KUKA KRL program: EPS_2_25694_SR02_A_20251117072413.src

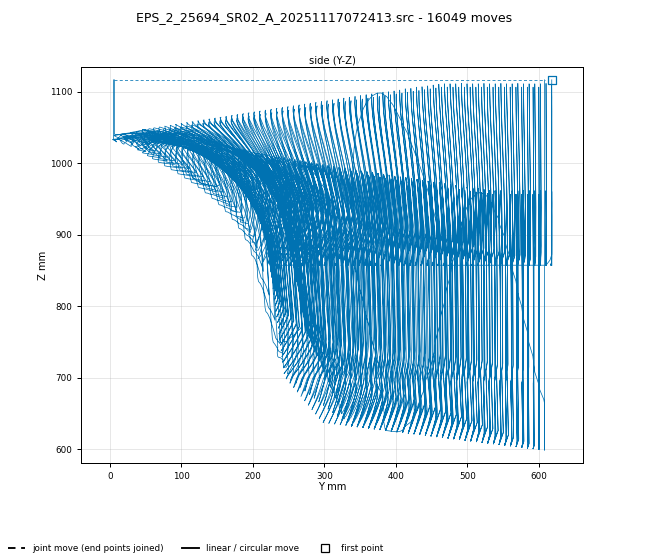
[picture p0: tool path of EPS_2_25694_SR02_A_20251117072413.src, 16049 of 16051 moves have a stored position in this frame; points joined in program order, loops and branches not executed]
&ACCESS RVP
&REL 4
&COMMENT QRS 19112012
&PARAM EDITMASK = *
DEF PART()
EXT BAS (BAS_COMMAND :IN,REAL :IN )
INT I
BAS (#INITMOV,0 )

;KUKA QRS Post kuka4.cps  Date:22-06-2017 !

File_ID=2907

QRS_PRE_INIT()

;Init var - Until changes are made in qrs_pre_init
Outlet_Square_prg=0
Inlet_1_Square_prg=0
Inlet_2_Square_prg=0
Inlet_3_Square_prg=0
Inlet_4_Square_prg=0
Inlet_5_Square_prg=0

Outlet_1={X 0.000, Y 466.000, Z 916.000, B 0.000, E1 0.000 }
Inlet_1={X 0.000, Y 530.840, Z 461.000, B 0.000, E1 112.000 }
Inlet_2={X 0.000, Y 532.280, Z 441.000, B 0.000, E1 197.000 }
Outlet_1_type=381
Inlet_1_type=251
Inlet_2_type=251
;QRS#1=Sidecore dimensions
;QRS#2=375-15" Concrete
;QRS#3=250-10" PVC SDR 35
;QRS#4=250-10" PVC SDR 35
;QRS#5=
;QRS#6=
;QRS#7=
;QRS#8=
;QRS#9=24L PSX-2
;QRS#10=14M PSX
;QRS#11=14M PSX
;QRS#12=
;QRS#13=
;QRS#14=
;QRS#15=
;QRS#16=1220x127x1448 4,75'
;QRS#17=EPS Height
;QRS#18=1106,5
;QRS#19=*
;QRS#20= UPDATED VERSION 22-06-2017
;QRS#21=*
Outlet_Square=0150
Inlet_1_Square=0100
Inlet_2_Square=0100
Inlet_3_Square=0
Inlet_4_Square=0
Inlet_5_Square=0
Mill_Square=1
Outlet_Square_Prg=261
Inlet_1_Square_prg=205
Inlet_2_Square_prg=205

QRS_INIT()

$ADVANCE=5

; T1
PTP {E1 171.09,E2 171.09}
PTP {X 0,Y 618.04,A -85,B 0,C 180,E1 171.09,E2 171.09,E3 0,E4 0,E5 0,E6 0}
QRS_SPEED_INIT()
LIN {X 0,Y 618.04,Z 1116.5,A -85,B 0,C 180,E1 171.09,E2 171.09,E3 0,E4 0,E5 0,E6 0} C_VEL
LIN {X 0,Y 618.04,Z 893.453,A -85,B 0,C 180,E1 171.09,E2 171.09} C_VEL
LIN {X 0,Y 618.04,Z 872.961,A -85,B 0,C 180,E1 171.09,E2 171.09} C_VEL
LIN {X 0,Y 618.039,Z 872.148,A -85,B 0,C 180,E1 171.106,E2 171.106} C_VEL
LIN {X 0,Y 618.037,Z 863.35,A -85,B 0,C 180,E1 171.469,E2 171.469} C_VEL
LIN {X 0,Y 617.988,Z 857.28,A -85,B 0,C 180,E1 171.692,E2 171.692} C_VEL
LIN {X 0,Y 618.064,Z 857.28,A -85,B 0,C 180,E1 171.887,E2 171.887} C_VEL
LIN {X 0,Y 618.025,Z 857.28,A -85,B 0,C 180,E1 174.214,E2 174.214} C_VEL
LIN {X 0,Y 618.042,Z 857.28,A -85,B 0,C 180,E1 178.845,E2 178.845} C_VEL
LIN {X 0,Y 618.069,Z 857.28,A -85,B 0,C 180,E1 183.468,E2 183.468} C_VEL
LIN {X 0,Y 618.042,Z 857.28,A -85,B 0,C 180,E1 188.114,E2 188.114} C_VEL
LIN {X 0,Y 617.972,Z 857.28,A -85,B 0,C 180,E1 192.816,E2 192.816} C_VEL
LIN {X 0,Y 617.962,Z 857.28,A -85,B 0,C 180,E1 197.607,E2 197.607} C_VEL
LIN {X 0,Y 617.779,Z 857.28,A -85,B 0,C 180,E1 198.55,E2 198.55} C_VEL
LIN {X 0,Y 617.956,Z 857.28,A -85,B 0,C 180,E1 202.529,E2 202.529} C_VEL
LIN {X 0,Y 617.453,Z 857.28,A -85,B 0,C 180,E1 205.076,E2 205.076} C_VEL
LIN {X 0,Y 617.89,Z 857.28,A -85,B 0,C 180,E1 207.636,E2 207.636} C_VEL
LIN {X 0,Y 617.381,Z 857.28,A -85,B 0,C 180,E1 210.305,E2 210.305} C_VEL
LIN {X 0,Y 617.848,Z 857.28,A -85,B 0,C 180,E1 212.995,E2 212.995} C_VEL
LIN {X 0,Y 617.72,Z 857.28,A -85,B 0,C 180,E1 214.198,E2 214.198} C_VEL
LIN {X 0,Y 617.794,Z 857.28,A -85,B 0,C 180,E1 218.704,E2 218.704} C_VEL
LIN {X 0,Y 617.454,Z 857.28,A -85,B 0,C 180,E1 221.759,E2 221.759} C_VEL
LIN {X 0,Y 617.88,Z 857.28,A -85,B 0,C 180,E1 224.901,E2 224.901} C_VEL
LIN {X 0,Y 617.78,Z 857.28,A -85,B 0,C 180,E1 228.274,E2 228.274} C_VEL
LIN {X 0,Y 617.552,Z 857.28,A -85,B 0,C 180,E1 231.278,E2 231.278} C_VEL
LIN {X 0,Y 617.574,Z 857.28,A -85,B 0,C 180,E1 231.9,E2 231.9} C_VEL
LIN {X 0,Y 617.805,Z 857.28,A -85,B 0,C 180,E1 234.201,E2 234.201} C_VEL
LIN {X 0,Y 617.346,Z 857.28,A -85,B 0,C 180,E1 236.975,E2 236.975} C_VEL
LIN {X 0,Y 617.903,Z 857.28,A -85,B 0,C 180,E1 239.723,E2 239.723} C_VEL
LIN {X 0,Y 617.426,Z 857.28,A -85,B 0,C 180,E1 242.341,E2 242.341} C_VEL
LIN {X 0,Y 617.95,Z 857.28,A -85,B 0,C 180,E1 244.946,E2 244.946} C_VEL
LIN {X 0,Y 617.971,Z 857.28,A -85,B 0,C 180,E1 247.993,E2 247.993} C_VEL
LIN {X 0,Y 617.845,Z 857.28,A -85,B 0,C 180,E1 248.248,E2 248.248} C_VEL
LIN {X 0,Y 616.597,Z 857.28,A -85,B 0,C 180,E1 248.461,E2 248.461} C_VEL
LIN {X 0,Y 617.498,Z 860.533,A -85,B 0,C 180,E1 248.542,E2 248.542} C_VEL
LIN {X 0,Y 617.689,Z 861.463,A -85,B 0,C 180,E1 248.56,E2 248.56} C_VEL
LIN {X 0,Y 617.924,Z 919.311,A -85,B 0,C 180,E1 249.277,E2 249.277} C_VEL
LIN {X 0,Y 618.001,Z 930.791,A -85,B 0,C 180,E1 249.459,E2 249.459} C_VEL
LIN {X 0,Y 617.956,Z 939.703,A -85,B 0,C 180,E1 249.638,E2 249.638} C_VEL
LIN {X 0,Y 617.868,Z 948.851,A -85,B 0,C 180,E1 249.859,E2 249.859} C_VEL
LIN {X 0,Y 617.969,Z 959.233,A -85,B 0,C 180,E1 250.169,E2 250.169} C_VEL
LIN {X 0,Y 617.951,Z 969.224,A -85,B 0,C 180,E1 250.516,E2 250.516} C_VEL
LIN {X 0,Y 617.933,Z 976.981,A -85,B 0,C 180,E1 250.818,E2 250.818} C_VEL
LIN {X 0,Y 617.992,Z 986.692,A -85,B 0,C 180,E1 251.252,E2 251.252} C_VEL
LIN {X 0,Y 618.003,Z 996.669,A -85,B 0,C 180,E1 251.755,E2 251.755} C_VEL
LIN {X 0,Y 617.953,Z 1005.465,A -85,B 0,C 180,E1 252.248,E2 252.248} C_VEL
LIN {X 0,Y 617.994,Z 1014.291,A -85,B 0,C 180,E1 252.801,E2 252.801} C_VEL
LIN {X 0,Y 617.978,Z 1023.074,A -85,B 0,C 180,E1 253.409,E2 253.409} C_VEL
LIN {X 0,Y 617.993,Z 1031.008,A -85,B 0,C 180,E1 254.015,E2 254.015} C_VEL
LIN {X 0,Y 617.98,Z 1038.115,A -85,B 0,C 180,E1 254.606,E2 254.606} C_VEL
LIN {X 0,Y 617.953,Z 1043.662,A -85,B 0,C 180,E1 255.101,E2 255.101} C_VEL
LIN {X 0,Y 617.981,Z 1051.279,A -85,B 0,C 180,E1 255.848,E2 255.848} C_VEL
LIN {X 0,Y 618.005,Z 1056.878,A -85,B 0,C 180,E1 256.443,E2 256.443} C_VEL
LIN {X 0,Y 617.937,Z 1063.299,A -85,B 0,C 180,E1 257.184,E2 257.184} C_VEL
LIN {X 0,Y 617.922,Z 1069.145,A -85,B 0,C 180,E1 257.923,E2 257.923} C_VEL
LIN {X 0,Y 617.97,Z 1074.465,A -85,B 0,C 180,E1 258.661,E2 258.661} C_VEL
LIN {X 0,Y 617.959,Z 1080.218,A -85,B 0,C 180,E1 259.544,E2 259.544} C_VEL
LIN {X 0,Y 617.879,Z 1084.857,A -85,B 0,C 180,E1 260.327,E2 260.327} C_VEL
LIN {X 0,Y 617.887,Z 1089.451,A -85,B 0,C 180,E1 261.196,E2 261.196} C_VEL
LIN {X 0,Y 617.977,Z 1093.733,A -85,B 0,C 180,E1 262.119,E2 262.119} C_VEL
LIN {X 0,Y 617.893,Z 1096.689,A -85,B 0,C 180,E1 262.817,E2 262.817} C_VEL
LIN {X 0,Y 617.823,Z 1100.1,A -85,B 0,C 180,E1 263.747,E2 263.747} C_VEL
LIN {X 0,Y 617.905,Z 1102.963,A -85,B 0,C 180,E1 264.677,E2 264.677} C_VEL
LIN {X 0,Y 617.95,Z 1105.345,A -85,B 0,C 180,E1 265.605,E2 265.605} C_VEL
LIN {X 0,Y 617.834,Z 1107.293,A -85,B 0,C 180,E1 266.531,E2 266.531} C_VEL
LIN {X 0,Y 617.839,Z 1108.744,A -85,B 0,C 180,E1 267.457,E2 267.457} C_VEL
LIN {X 0,Y 617.944,Z 1110.042,A -85,B 0,C 180,E1 268.845,E2 268.845} C_VEL
LIN {X 0,Y 617.878,Z 1110.288,A -85,B 0,C 180,E1 269.307,E2 269.307} C_VEL
LIN {X 0,Y 617.832,Z 1110.409,A -85,B 0,C 180,E1 270.231,E2 270.231} C_VEL
LIN {X 0,Y 617.902,Z 1110.053,A -85,B 0,C 180,E1 271.156,E2 271.156} C_VEL
LIN {X 0,Y 617.951,Z 1109.26,A -85,B 0,C 180,E1 272.08,E2 272.08} C_VEL
LIN {X 0,Y 617.822,Z 1107.296,A -85,B 0,C 180,E1 273.469,E2 273.469} C_VEL
LIN {X 0,Y 617.899,Z 1105.359,A -85,B 0,C 180,E1 274.395,E2 274.395} C_VEL
LIN {X 0,Y 617.943,Z 1102.953,A -85,B 0,C 180,E1 275.323,E2 275.323} C_VEL
LIN {X 0,Y 617.836,Z 1100.097,A -85,B 0,C 180,E1 276.253,E2 276.253} C_VEL
LIN {X 0,Y 617.864,Z 1096.696,A -85,B 0,C 180,E1 277.183,E2 277.183} C_VEL
LIN {X 0,Y 617.981,Z 1091.704,A -85,B 0,C 180,E1 278.334,E2 278.334} C_VEL
LIN {X 0,Y 617.877,Z 1086.888,A -85,B 0,C 180,E1 279.301,E2 279.301} C_VEL
LIN {X 0,Y 617.884,Z 1082.576,A -85,B 0,C 180,E1 280.072,E2 280.072} C_VEL
LIN {X 0,Y 617.947,Z 1078.418,A -85,B 0,C 180,E1 280.751,E2 280.751} C_VEL
LIN {X 0,Y 617.962,Z 1072.408,A -85,B 0,C 180,E1 281.634,E2 281.634} C_VEL
LIN {X 0,Y 617.908,Z 1065.701,A -85,B 0,C 180,E1 282.521,E2 282.521} C_VEL
LIN {X 0,Y 617.947,Z 1059.514,A -85,B 0,C 180,E1 283.261,E2 283.261} C_VEL
LIN {X 0,Y 617.996,Z 1054.147,A -85,B 0,C 180,E1 283.854,E2 283.854} C_VEL
LIN {X 0,Y 617.97,Z 1046.794,A -85,B 0,C 180,E1 284.6,E2 284.6} C_VEL
LIN {X 0,Y 617.961,Z 1040.369,A -85,B 0,C 180,E1 285.198,E2 285.198} C_VEL
LIN {X 0,Y 617.985,Z 1032.107,A -85,B 0,C 180,E1 285.897,E2 285.897} C_VEL
LIN {X 0,Y 617.995,Z 1024.024,A -85,B 0,C 180,E1 286.521,E2 286.521} C_VEL
LIN {X 0,Y 617.984,Z 1016.498,A -85,B 0,C 180,E1 287.052,E2 287.052} C_VEL
LIN {X 0,Y 617.987,Z 1009.682,A -85,B 0,C 180,E1 287.495,E2 287.495} C_VEL
LIN {X 0,Y 617.943,Z 1001.121,A -85,B 0,C 180,E1 288.003,E2 288.003} C_VEL
LIN {X 0,Y 617.999,Z 992.467,A -85,B 0,C 180,E1 288.464,E2 288.464} C_VEL
LIN {X 0,Y 618.009,Z 982.893,A -85,B 0,C 180,E1 288.921,E2 288.921} C_VEL
LIN {X 0,Y 617.967,Z 973.713,A -85,B 0,C 180,E1 289.311,E2 289.311} C_VEL
LIN {X 0,Y 617.906,Z 965.71,A -85,B 0,C 180,E1 289.616,E2 289.616} C_VEL
LIN {X 0,Y 618.002,Z 954.078,A -85,B 0,C 180,E1 289.987,E2 289.987} C_VEL
LIN {X 0,Y 617.983,Z 944.339,A -85,B 0,C 180,E1 290.251,E2 290.251} C_VEL
LIN {X 0,Y 617.847,Z 934.408,A -85,B 0,C 180,E1 290.477,E2 290.477} C_VEL
LIN {X 0,Y 617.928,Z 924.756,A -85,B 0,C 180,E1 290.644,E2 290.644} C_VEL
LIN {X 0,Y 617.881,Z 903.608,A -85,B 0,C 180,E1 290.919,E2 290.919} C_VEL
LIN {X 0,Y 617.753,Z 864.651,A -85,B 0,C 180,E1 291.399,E2 291.399} C_VEL
LIN {X 0,Y 617.582,Z 861.01,A -85,B 0,C 180,E1 291.45,E2 291.45} C_VEL
LIN {X 0,Y 616.602,Z 857.28,A -85,B 0,C 180,E1 291.54,E2 291.54} C_VEL
LIN {X 0,Y 618.005,Z 857.28,A -85,B 0,C 180,E1 291.926,E2 291.926} C_VEL
LIN {X 0,Y 618.025,Z 857.28,A -85,B 0,C 180,E1 292.526,E2 292.526} C_VEL
LIN {X 0,Y 617.436,Z 857.28,A -85,B 0,C 180,E1 295.077,E2 295.077} C_VEL
LIN {X 0,Y 617.88,Z 857.28,A -85,B 0,C 180,E1 297.637,E2 297.637} C_VEL
LIN {X 0,Y 617.376,Z 857.28,A -85,B 0,C 180,E1 300.306,E2 300.306} C_VEL
LIN {X 0,Y 617.847,Z 857.28,A -85,B 0,C 180,E1 302.995,E2 302.995} C_VEL
LIN {X 0,Y 617.71,Z 857.28,A -85,B 0,C 180,E1 304.197,E2 304.197} C_VEL
LIN {X 0,Y 617.806,Z 857.28,A -85,B 0,C 180,E1 308.703,E2 308.703} C_VEL
LIN {X 0,Y 617.453,Z 857.28,A -85,B 0,C 180,E1 311.759,E2 311.759} C_VEL
LIN {X 0,Y 617.865,Z 857.28,A -85,B 0,C 180,E1 314.902,E2 314.902} C_VEL
LIN {X 0,Y 617.768,Z 857.28,A -85,B 0,C 180,E1 318.275,E2 318.275} C_VEL
LIN {X 0,Y 617.555,Z 857.28,A -85,B 0,C 180,E1 321.279,E2 321.279} C_VEL
LIN {X 0,Y 617.591,Z 857.28,A -85,B 0,C 180,E1 321.898,E2 321.898} C_VEL
LIN {X 0,Y 617.836,Z 857.28,A -85,B 0,C 180,E1 324.203,E2 324.203} C_VEL
LIN {X 0,Y 617.346,Z 857.28,A -85,B 0,C 180,E1 326.975,E2 326.975} C_VEL
LIN {X 0,Y 617.862,Z 857.28,A -85,B 0,C 180,E1 329.721,E2 329.721} C_VEL
LIN {X 0,Y 617.414,Z 857.28,A -85,B 0,C 180,E1 332.341,E2 332.341} C_VEL
LIN {X 0,Y 617.92,Z 857.28,A -85,B 0,C 180,E1 334.944,E2 334.944} C_VEL
LIN {X 0,Y 617.455,Z 857.28,A -85,B 0,C 180,E1 337.452,E2 337.452} C_VEL
LIN {X 0,Y 617.949,Z 857.28,A -85,B 0,C 180,E1 339.951,E2 339.951} C_VEL
LIN {X 0,Y 618.039,Z 857.28,A -85,B 0,C 180,E1 343.632,E2 343.632} C_VEL
LIN {X 0,Y 618.002,Z 857.28,A -85,B 0,C 180,E1 349.544,E2 349.544} C_VEL
LIN {X 0,Y 618.032,Z 857.28,A -85,B 0,C 180,E1 354.214,E2 354.214} C_VEL
LIN {X 0,Y 618.053,Z 857.28,A -85,B 0,C 180,E1 358.845,E2 358.845} C_VEL
LIN {X 0,Y 618.057,Z 857.28,A -85,B 0,C 180,E1 363.468,E2 363.468} C_VEL
LIN {X 0,Y 618.041,Z 857.28,A -85,B 0,C 180,E1 368.114,E2 368.114} C_VEL
LIN {X 0,Y 617.985,Z 857.28,A -85,B 0,C 180,E1 372.815,E2 372.815} C_VEL
LIN {X 0,Y 617.978,Z 857.28,A -85,B 0,C 180,E1 377.606,E2 377.606} C_VEL
LIN {X 0,Y 617.784,Z 857.28,A -85,B 0,C 180,E1 378.551,E2 378.551} C_VEL
LIN {X 0,Y 617.941,Z 857.28,A -85,B 0,C 180,E1 382.529,E2 382.529} C_VEL
LIN {X 0,Y 617.448,Z 857.28,A -85,B 0,C 180,E1 385.076,E2 385.076} C_VEL
LIN {X 0,Y 617.897,Z 857.28,A -85,B 0,C 180,E1 387.636,E2 387.636} C_VEL
LIN {X 0,Y 617.383,Z 857.28,A -85,B 0,C 180,E1 390.305,E2 390.305} C_VEL
LIN {X 0,Y 617.849,Z 857.28,A -85,B 0,C 180,E1 392.995,E2 392.995} C_VEL
LIN {X 0,Y 617.708,Z 857.28,A -85,B 0,C 180,E1 394.196,E2 394.196} C_VEL
LIN {X 0,Y 617.785,Z 857.28,A -85,B 0,C 180,E1 398.704,E2 398.704} C_VEL
LIN {X 0,Y 617.446,Z 857.28,A -85,B 0,C 180,E1 401.76,E2 401.76} C_VEL
LIN {X 0,Y 617.879,Z 857.28,A -85,B 0,C 180,E1 404.901,E2 404.901} C_VEL
LIN {X 0,Y 617.763,Z 857.28,A -85,B 0,C 180,E1 408.276,E2 408.276} C_VEL
LIN {X 0,Y 617.554,Z 857.28,A -85,B 0,C 180,E1 411.278,E2 411.278} C_VEL
LIN {X 0,Y 617.581,Z 857.28,A -85,B 0,C 180,E1 411.9,E2 411.9} C_VEL
LIN {X 0,Y 617.842,Z 857.28,A -85,B 0,C 180,E1 414.204,E2 414.204} C_VEL
LIN {X 0,Y 618.036,Z 857.28,A -85,B 0,C 180,E1 418.887,E2 418.887} C_VEL
LIN {X 0,Y 618.021,Z 857.28,A -85,B 0,C 180,E1 419.078,E2 419.078} C_VEL
LIN {X 0,Y 617.565,Z 857.357,A -85,B 0,C 180,E1 419.213,E2 419.213} C_VEL
LIN {X 0,Y 617.922,Z 866.552,A -85,B 0,C 180,E1 419.562,E2 419.562} C_VEL
LIN {X 0,Y 617.999,Z 875.408,A -85,B 0,C 180,E1 419.958,E2 419.958} C_VEL
LIN {X 0,Y 617.995,Z 884.21,A -85,B 0,C 180,E1 420.411,E2 420.411} C_VEL
LIN {X 0,Y 618.021,Z 891.714,A -85,B 0,C 180,E1 420.859,E2 420.859} C_VEL
LIN {X 0,Y 618.016,Z 898.437,A -85,B 0,C 180,E1 421.312,E2 421.312} C_VEL
LIN {X 0,Y 618.01,Z 905.925,A -85,B 0,C 180,E1 421.877,E2 421.877} C_VEL
LIN {X 0,Y 617.989,Z 913.549,A -85,B 0,C 180,E1 422.532,E2 422.532} C_VEL
LIN {X 0,Y 617.986,Z 920.183,A -85,B 0,C 180,E1 423.181,E2 423.181} C_VEL
LIN {X 0,Y 617.987,Z 927.401,A -85,B 0,C 180,E1 423.987,E2 423.987} C_VEL
LIN {X 0,Y 617.977,Z 932.435,A -85,B 0,C 180,E1 424.627,E2 424.627} C_VEL
LIN {X 0,Y 617.963,Z 937.67,A -85,B 0,C 180,E1 425.376,E2 425.376} C_VEL
LIN {X 0,Y 617.994,Z 942.305,A -85,B 0,C 180,E1 426.144,E2 426.144} C_VEL
LIN {X 0,Y 617.943,Z 946.382,A -85,B 0,C 180,E1 426.92,E2 426.92} C_VEL
LIN {X 0,Y 617.93,Z 950.266,A -85,B 0,C 180,E1 427.783,E2 427.783} C_VEL
LIN {X 0,Y 617.999,Z 953.633,A -85,B 0,C 180,E1 428.718,E2 428.718} C_VEL
LIN {X 0,Y 617.953,Z 955.499,A -85,B 0,C 180,E1 429.335,E2 429.335} C_VEL
LIN {X 0,Y 617.897,Z 957.055,A -85,B 0,C 180,E1 429.95,E2 429.95} C_VEL
LIN {X 0,Y 617.918,Z 958.426,A -85,B 0,C 180,E1 430.644,E2 430.644} C_VEL
LIN {X 0,Y 617.988,Z 959.481,A -85,B 0,C 180,E1 431.393,E2 431.393} C_VEL
LIN {X 0,Y 617.929,Z 960.308,A -85,B 0,C 180,E1 432.392,E2 432.392} C_VEL
LIN {X 0,Y 617.908,Z 960.363,A -85,B 0,C 180,E1 433.299,E2 433.299} C_VEL
LIN {X 0,Y 617.931,Z 960.207,A -85,B 0,C 180,E1 433.707,E2 433.707} C_VEL
LIN {X 0,Y 617.953,Z 959.156,A -85,B 0,C 180,E1 434.802,E2 434.802} C_VEL
LIN {X 0,Y 617.917,Z 958.206,A -85,B 0,C 180,E1 435.399,E2 435.399} C_VEL
LIN {X 0,Y 617.92,Z 956.973,A -85,B 0,C 180,E1 435.995,E2 435.995} C_VEL
LIN {X 0,Y 617.963,Z 955.452,A -85,B 0,C 180,E1 436.591,E2 436.591} C_VEL
LIN {X 0,Y 617.974,Z 952.698,A -85,B 0,C 180,E1 437.48,E2 437.48} C_VEL
LIN {X 0,Y 617.922,Z 950.503,A -85,B 0,C 180,E1 438.071,E2 438.071} C_VEL
LIN {X 0,Y 617.922,Z 947.977,A -85,B 0,C 180,E1 438.66,E2 438.66} C_VEL
LIN {X 0,Y 617.993,Z 943.521,A -85,B 0,C 180,E1 439.544,E2 439.544} C_VEL
LIN {X 0,Y 617.983,Z 939.081,A -85,B 0,C 180,E1 440.309,E2 440.309} C_VEL
LIN {X 0,Y 617.958,Z 933.399,A -85,B 0,C 180,E1 441.154,E2 441.154} C_VEL
LIN {X 0,Y 617.993,Z 927.705,A -85,B 0,C 180,E1 441.886,E2 441.886} C_VEL
LIN {X 0,Y 618.001,Z 921.58,A -85,B 0,C 180,E1 442.585,E2 442.585} C_VEL
LIN {X 0,Y 617.982,Z 915.8,A -85,B 0,C 180,E1 443.167,E2 443.167} C_VEL
LIN {X 0,Y 618.005,Z 909.346,A -85,B 0,C 180,E1 443.749,E2 443.749} C_VEL
LIN {X 0,Y 618.016,Z 902.149,A -85,B 0,C 180,E1 444.33,E2 444.33} C_VEL
LIN {X 0,Y 618.029,Z 893.855,A -85,B 0,C 180,E1 444.91,E2 444.91} C_VEL
LIN {X 0,Y 618.019,Z 886.367,A -85,B 0,C 180,E1 445.374,E2 445.374} C_VEL
LIN {X 0,Y 618.034,Z 877.771,A -85,B 0,C 180,E1 445.837,E2 445.837} C_VEL
LIN {X 0,Y 618.041,Z 868.943,A -85,B 0,C 180,E1 446.243,E2 446.243} C_VEL
LIN {X 0,Y 618.015,Z 860.032,A -85,B 0,C 180,E1 446.594,E2 446.594} C_VEL
LIN {X 0,Y 617.985,Z 857.28,A -85,B 0,C 180,E1 446.693,E2 446.693} C_VEL
LIN {X 0,Y 618.049,Z 857.28,A -85,B 0,C 180,E1 447.468,E2 447.468} C_VEL
LIN {X 0,Y 617.305,Z 857.28,A -85,B 0,C 180,E1 451.157,E2 451.157} C_VEL
LIN {X 0,Y 618.059,Z 857.28,A -85,B 0,C 180,E1 453.468,E2 453.468} C_VEL
LIN {X 0,Y 618.052,Z 857.28,A -85,B 0,C 180,E1 458.114,E2 458.114} C_VEL
LIN {X 0,Y 618.016,Z 857.28,A -85,B 0,C 180,E1 462.815,E2 462.815} C_VEL
LIN {X 0,Y 617.938,Z 857.28,A -85,B 0,C 180,E1 467.607,E2 467.607} C_VEL
LIN {X 0,Y 617.759,Z 857.28,A -85,B 0,C 180,E1 468.544,E2 468.544} C_VEL
LIN {X 0,Y 617.93,Z 857.28,A -85,B 0,C 180,E1 472.53,E2 472.53} C_VEL
LIN {X 0,Y 617.424,Z 857.28,A -85,B 0,C 180,E1 475.077,E2 475.077} C_VEL
LIN {X 0,Y 617.857,Z 857.28,A -85,B 0,C 180,E1 477.638,E2 477.638} C_VEL
LIN {X 0,Y 617.361,Z 857.28,A -85,B 0,C 180,E1 480.306,E2 480.306} C_VEL
LIN {X 0,Y 617.851,Z 857.28,A -85,B 0,C 180,E1 482.995,E2 482.995} C_VEL
LIN {X 0,Y 617.718,Z 857.28,A -85,B 0,C 180,E1 484.198,E2 484.198} C_VEL
LIN {X 0,Y 617.747,Z 857.28,A -85,B 0,C 180,E1 488.707,E2 488.707} C_VEL
LIN {X 0,Y 617.425,Z 857.28,A -85,B 0,C 180,E1 491.762,E2 491.762} C_VEL
LIN {X 0,Y 617.878,Z 857.28,A -85,B 0,C 180,E1 494.901,E2 494.901} C_VEL
LIN {X 0,Y 617.786,Z 857.28,A -85,B 0,C 180,E1 498.273,E2 498.273} C_VEL
LIN {X 0,Y 617.488,Z 857.28,A -85,B 0,C 180,E1 501.274,E2 501.274} C_VEL
LIN {X 0,Y 617.755,Z 857.299,A -85,B 0,C 180,E1 504.216,E2 504.216} C_VEL
LIN {X 0,Y 617.946,Z 867.414,A -85,B 0,C 180,E1 504.599,E2 504.599} C_VEL
LIN {X 0,Y 617.985,Z 875.042,A -85,B 0,C 180,E1 504.94,E2 504.94} C_VEL
LIN {X 0,Y 618.02,Z 883.242,A -85,B 0,C 180,E1 505.36,E2 505.36} C_VEL
LIN {X 0,Y 618.032,Z 892.212,A -85,B 0,C 180,E1 505.892,E2 505.892} C_VEL
LIN {X 0,Y 617.997,Z 899.299,A -85,B 0,C 180,E1 506.373,E2 506.373} C_VEL
LIN {X 0,Y 618.002,Z 905.644,A -85,B 0,C 180,E1 506.855,E2 506.855} C_VEL
LIN {X 0,Y 618.008,Z 913.37,A -85,B 0,C 180,E1 507.515,E2 507.515} C_VEL
LIN {X 0,Y 617.992,Z 919.727,A -85,B 0,C 180,E1 508.134,E2 508.134} C_VEL
LIN {X 0,Y 617.968,Z 926.591,A -85,B 0,C 180,E1 508.887,E2 508.887} C_VEL
LIN {X 0,Y 617.959,Z 931.93,A -85,B 0,C 180,E1 509.559,E2 509.559} C_VEL
LIN {X 0,Y 617.992,Z 937.196,A -85,B 0,C 180,E1 510.307,E2 510.307} C_VEL
LIN {X 0,Y 617.969,Z 941.404,A -85,B 0,C 180,E1 510.982,E2 510.982} C_VEL
LIN {X 0,Y 617.919,Z 945.817,A -85,B 0,C 180,E1 511.802,E2 511.802} C_VEL
LIN {X 0,Y 617.987,Z 949.867,A -85,B 0,C 180,E1 512.694,E2 512.694} C_VEL
LIN {X 0,Y 617.938,Z 953.473,A -85,B 0,C 180,E1 513.663,E2 513.663} C_VEL
LIN {X 0,Y 617.908,Z 955.428,A -85,B 0,C 180,E1 514.304,E2 514.304} C_VEL
LIN {X 0,Y 617.954,Z 957.484,A -85,B 0,C 180,E1 515.155,E2 515.155} C_VEL
LIN {X 0,Y 618.001,Z 958.389,A -85,B 0,C 180,E1 515.636,E2 515.636} C_VEL
LIN {X 0,Y 617.94,Z 959.543,A -85,B 0,C 180,E1 516.434,E2 516.434} C_VEL
LIN {X 0,Y 617.921,Z 960.327,A -85,B 0,C 180,E1 517.47,E2 517.47} C_VEL
LIN {X 0,Y 617.975,Z 960.393,A -85,B 0,C 180,E1 518.096,E2 518.096} C_VEL
LIN {X 0,Y 617.968,Z 960.189,A -85,B 0,C 180,E1 518.717,E2 518.717} C_VEL
LIN {X 0,Y 617.943,Z 959.71,A -85,B 0,C 180,E1 519.335,E2 519.335} C_VEL
LIN {X 0,Y 617.929,Z 958.95,A -85,B 0,C 180,E1 519.951,E2 519.951} C_VEL
LIN {X 0,Y 617.992,Z 957.697,A -85,B 0,C 180,E1 520.652,E2 520.652} C_VEL
LIN {X 0,Y 617.962,Z 955.964,A -85,B 0,C 180,E1 521.4,E2 521.4} C_VEL
LIN {X 0,Y 617.917,Z 954.689,A -85,B 0,C 180,E1 521.87,E2 521.87} C_VEL
LIN {X 0,Y 617.91,Z 953.019,A -85,B 0,C 180,E1 522.392,E2 522.392} C_VEL
LIN {X 0,Y 617.957,Z 949.943,A -85,B 0,C 180,E1 523.2,E2 523.2} C_VEL
LIN {X 0,Y 617.982,Z 946.308,A -85,B 0,C 180,E1 524.003,E2 524.003} C_VEL
LIN {X 0,Y 617.988,Z 942.107,A -85,B 0,C 180,E1 524.803,E2 524.803} C_VEL
LIN {X 0,Y 617.96,Z 938.532,A -85,B 0,C 180,E1 525.4,E2 525.4} C_VEL
LIN {X 0,Y 617.959,Z 933.465,A -85,B 0,C 180,E1 526.145,E2 526.145} C_VEL
LIN {X 0,Y 617.998,Z 927.679,A -85,B 0,C 180,E1 526.889,E2 526.889} C_VEL
LIN {X 0,Y 617.992,Z 921.164,A -85,B 0,C 180,E1 527.629,E2 527.629} C_VEL
LIN {X 0,Y 617.991,Z 915.241,A -85,B 0,C 180,E1 528.219,E2 528.219} C_VEL
LIN {X 0,Y 618.018,Z 908.638,A -85,B 0,C 180,E1 528.809,E2 528.809} C_VEL
LIN {X 0,Y 618.03,Z 900.192,A -85,B 0,C 180,E1 529.471,E2 529.471} C_VEL
LIN {X 0,Y 618.017,Z 893.812,A -85,B 0,C 180,E1 529.913,E2 529.913} C_VEL
LIN {X 0,Y 618.003,Z 886.379,A -85,B 0,C 180,E1 530.374,E2 530.374} C_VEL
LIN {X 0,Y 618.037,Z 877.84,A -85,B 0,C 180,E1 530.834,E2 530.834} C_VEL
LIN {X 0,Y 618.039,Z 872.148,A -85,B 0,C 180,E1 531.106,E2 531.106} C_VEL
LIN {X 0,Y 615.518,Z 864.313,A -85,B 0,C 180,E1 531.544,E2 531.544} C_VEL
LIN {X 0,Y 610.896,Z 858.156,A -85,B 0,C 180,E1 532.238,E2 532.238} C_VEL
LIN {X 0,Y 610.06,Z 857.28,A -85,B 0,C 180,E1 532.633,E2 532.633} C_VEL
LIN {X 0,Y 610.057,Z 857.28,A -85,B 0,C 180,E1 538.597,E2 538.597} C_VEL
LIN {X 0,Y 609.894,Z 857.28,A -85,B 0,C 180,E1 544.287,E2 544.287} C_VEL
LIN {X 0,Y 609.957,Z 857.28,A -85,B 0,C 180,E1 548.58,E2 548.58} C_VEL
LIN {X 0,Y 610.038,Z 857.28,A -85,B 0,C 180,E1 552.92,E2 552.92} C_VEL
LIN {X 0,Y 609.816,Z 857.28,A -85,B 0,C 180,E1 558.841,E2 558.841} C_VEL
LIN {X 0,Y 609.758,Z 857.28,A -85,B 0,C 180,E1 563.418,E2 563.418} C_VEL
LIN {X 0,Y 609.804,Z 857.28,A -85,B 0,C 180,E1 568.155,E2 568.155} C_VEL
LIN {X 0,Y 609.954,Z 857.28,A -85,B 0,C 180,E1 573.105,E2 573.105} C_VEL
LIN {X 0,Y 609.619,Z 857.28,A -85,B 0,C 180,E1 579.653,E2 579.653} C_VEL
LIN {X 0,Y 609.739,Z 857.28,A -85,B 0,C 180,E1 585.951,E2 585.951} C_VEL
LIN {X 0,Y 609.56,Z 857.28,A -85,B 0,C 180,E1 590.353,E2 590.353} C_VEL
LIN {X 0,Y 609.597,Z 857.28,A -85,B 0,C 180,E1 595.163,E2 595.163} C_VEL
LIN {X 0,Y 609.798,Z 857.28,A -85,B 0,C 180,E1 600.338,E2 600.338} C_VEL
LIN {X 0,Y 610.046,Z 857.28,A -85,B 0,C 180,E1 605.044,E2 605.044} C_VEL
LIN {X 0,Y 609.377,Z 857.28,A -85,B 0,C 180,E1 608.167,E2 608.167} C_VEL
LIN {X 0,Y 610.37,Z 873.803,A -85,B 0,C 180,E1 608.443,E2 608.443} C_VEL
LIN {X 0,Y 610.561,Z 938.64,A -85,B 0,C 180,E1 609.354,E2 609.354} C_VEL
LIN {X 0,Y 610.451,Z 972.232,A -85,B 0,C 180,E1 610.384,E2 610.384} C_VEL
LIN {X 0,Y 610.386,Z 1004.124,A -85,B 0,C 180,E1 611.937,E2 611.937} C_VEL
LIN {X 0,Y 610.297,Z 1033.24,A -85,B 0,C 180,E1 613.979,E2 613.979} C_VEL
LIN {X 0,Y 610.237,Z 1058.073,A -85,B 0,C 180,E1 616.367,E2 616.367} C_VEL
LIN {X 0,Y 610.16,Z 1078.846,A -85,B 0,C 180,E1 619.094,E2 619.094} C_VEL
LIN {X 0,Y 610.159,Z 1095.118,A -85,B 0,C 180,E1 622.156,E2 622.156} C_VEL
LIN {X 0,Y 610.1,Z 1104.988,A -85,B 0,C 180,E1 625.018,E2 625.018} C_VEL
LIN {X 0,Y 610,Z 1109.397,A -85,B 0,C 180,E1 627.155,E2 627.155} C_VEL
LIN {X 0,Y 610.019,Z 1111.5,A -85,B 0,C 180,E1 630.001,E2 630.001} C_VEL
LIN {X 0,Y 610.048,Z 1109.396,A -85,B 0,C 180,E1 632.846,E2 632.846} C_VEL
LIN {X 0,Y 610.051,Z 1101.844,A -85,B 0,C 180,E1 636.056,E2 636.056} C_VEL
LIN {X 0,Y 610.116,Z 1090.12,A -85,B 0,C 180,E1 638.923,E2 638.923} C_VEL
LIN {X 0,Y 610.172,Z 1072.662,A -85,B 0,C 180,E1 641.813,E2 641.813} C_VEL
LIN {X 0,Y 610.233,Z 1050.188,A -85,B 0,C 180,E1 644.477,E2 644.477} C_VEL
LIN {X 0,Y 610.332,Z 1022.478,A -85,B 0,C 180,E1 646.855,E2 646.855} C_VEL
LIN {X 0,Y 610.439,Z 992.147,A -85,B 0,C 180,E1 648.717,E2 648.717} C_VEL
LIN {X 0,Y 610.516,Z 959.54,A -85,B 0,C 180,E1 650.073,E2 650.073} C_VEL
LIN {X 0,Y 610.548,Z 926.171,A -85,B 0,C 180,E1 650.885,E2 650.885} C_VEL
LIN {X 0,Y 609.709,Z 860.493,A -85,B 0,C 180,E1 651.747,E2 651.747} C_VEL
LIN {X 0,Y 609.512,Z 857.28,A -85,B 0,C 180,E1 651.877,E2 651.877} C_VEL
LIN {X 0,Y 609.659,Z 857.28,A -85,B 0,C 180,E1 656.622,E2 656.622} C_VEL
LIN {X 0,Y 609.95,Z 857.28,A -85,B 0,C 180,E1 663.101,E2 663.101} C_VEL
LIN {X 0,Y 609.607,Z 857.28,A -85,B 0,C 180,E1 669.653,E2 669.653} C_VEL
LIN {X 0,Y 609.706,Z 857.28,A -85,B 0,C 180,E1 675.946,E2 675.946} C_VEL
LIN {X 0,Y 609.561,Z 857.28,A -85,B 0,C 180,E1 680.355,E2 680.355} C_VEL
LIN {X 0,Y 609.624,Z 857.28,A -85,B 0,C 180,E1 685.159,E2 685.159} C_VEL
LIN {X 0,Y 609.747,Z 857.28,A -85,B 0,C 180,E1 690.354,E2 690.354} C_VEL
LIN {X 0,Y 609.999,Z 857.28,A -85,B 0,C 180,E1 695.033,E2 695.033} C_VEL
LIN {X 0,Y 609.8,Z 857.28,A -85,B 0,C 180,E1 701.158,E2 701.158} C_VEL
LIN {X 0,Y 609.378,Z 857.28,A -85,B 0,C 180,E1 705.7,E2 705.7} C_VEL
LIN {X 0,Y 609.94,Z 857.28,A -85,B 0,C 180,E1 709.979,E2 709.979} C_VEL
LIN {X 0,Y 610.117,Z 857.28,A -85,B 0,C 180,E1 714.287,E2 714.287} C_VEL
LIN {X 0,Y 609.785,Z 857.28,A -85,B 0,C 180,E1 719.982,E2 719.982} C_VEL
LIN {X 0,Y 609.874,Z 857.28,A -85,B 0,C 180,E1 724.251,E2 724.251} C_VEL
LIN {X 0,Y 609.97,Z 857.28,A -85,B 0,C 180,E1 728.543,E2 728.543} C_VEL
LIN {X 0,Y 610.049,Z 857.28,A -85,B 0,C 180,E1 732.883,E2 732.883} C_VEL
LIN {X 0,Y 609.808,Z 857.28,A -85,B 0,C 180,E1 738.803,E2 738.803} C_VEL
LIN {X 0,Y 609.739,Z 857.28,A -85,B 0,C 180,E1 743.379,E2 743.379} C_VEL
LIN {X 0,Y 609.807,Z 857.28,A -85,B 0,C 180,E1 748.114,E2 748.114} C_VEL
LIN {X 0,Y 609.933,Z 857.28,A -85,B 0,C 180,E1 753.063,E2 753.063} C_VEL
LIN {X 0,Y 609.617,Z 857.28,A -85,B 0,C 180,E1 759.651,E2 759.651} C_VEL
LIN {X 0,Y 609.731,Z 857.28,A -85,B 0,C 180,E1 765.949,E2 765.949} C_VEL
LIN {X 0,Y 609.556,Z 857.28,A -85,B 0,C 180,E1 770.296,E2 770.296} C_VEL
LIN {X 0,Y 609.656,Z 857.28,A -85,B 0,C 180,E1 775.165,E2 775.165} C_VEL
LIN {X 0,Y 609.909,Z 857.451,A -85,B 0,C 180,E1 779.036,E2 779.036} C_VEL
LIN {X 0,Y 610.278,Z 884.522,A -85,B 0,C 180,E1 780.251,E2 780.251} C_VEL
LIN {X 0,Y 610.245,Z 909.118,A -85,B 0,C 180,E1 781.962,E2 781.962} C_VEL
LIN {X 0,Y 610.185,Z 929.613,A -85,B 0,C 180,E1 784.065,E2 784.065} C_VEL
LIN {X 0,Y 610.147,Z 945.832,A -85,B 0,C 180,E1 786.554,E2 786.554} C_VEL
LIN {X 0,Y 610.156,Z 956.501,A -85,B 0,C 180,E1 789.291,E2 789.291} C_VEL
LIN {X 0,Y 610.141,Z 960.323,A -85,B 0,C 180,E1 791.179,E2 791.179} C_VEL
LIN {X 0,Y 610.098,Z 961.441,A -85,B 0,C 180,E1 792.674,E2 792.674} C_VEL
LIN {X 0,Y 610.11,Z 959.514,A -85,B 0,C 180,E1 795.263,E2 795.263} C_VEL
LIN {X 0,Y 610.148,Z 952.591,A -85,B 0,C 180,E1 797.823,E2 797.823} C_VEL
LIN {X 0,Y 610.182,Z 940.13,A -85,B 0,C 180,E1 800.357,E2 800.357} C_VEL
LIN {X 0,Y 610.208,Z 922.829,A -85,B 0,C 180,E1 802.636,E2 802.636} C_VEL
LIN {X 0,Y 610.27,Z 900.017,A -85,B 0,C 180,E1 804.661,E2 804.661} C_VEL
LIN {X 0,Y 610.366,Z 874.429,A -85,B 0,C 180,E1 806.177,E2 806.177} C_VEL
LIN {X 0,Y 610.123,Z 857.28,A -85,B 0,C 180,E1 806.888,E2 806.888} C_VEL
LIN {X 0,Y 609.888,Z 857.28,A -85,B 0,C 180,E1 814.271,E2 814.271} C_VEL
LIN {X 0,Y 609.965,Z 857.28,A -85,B 0,C 180,E1 818.565,E2 818.565} C_VEL
LIN {X 0,Y 610.08,Z 857.28,A -85,B 0,C 180,E1 822.906,E2 822.906} C_VEL
LIN {X 0,Y 609.793,Z 857.28,A -85,B 0,C 180,E1 828.831,E2 828.831} C_VEL
LIN {X 0,Y 609.716,Z 857.28,A -85,B 0,C 180,E1 833.41,E2 833.41} C_VEL
LIN {X 0,Y 609.768,Z 857.28,A -85,B 0,C 180,E1 838.149,E2 838.149} C_VEL
LIN {X 0,Y 609.954,Z 857.28,A -85,B 0,C 180,E1 843.099,E2 843.099} C_VEL
LIN {X 0,Y 609.549,Z 857.28,A -85,B 0,C 180,E1 849.703,E2 849.703} C_VEL
LIN {X 0,Y 609.737,Z 857.28,A -85,B 0,C 180,E1 855.999,E2 855.999} C_VEL
LIN {X 0,Y 609.528,Z 857.28,A -85,B 0,C 180,E1 860.357,E2 860.357} C_VEL
LIN {X 0,Y 609.855,Z 858,A -85,B 0,C 180,E1 864.053,E2 864.053} C_VEL
LIN {X 0,Y 610.318,Z 884.462,A -85,B 0,C 180,E1 865.248,E2 865.248} C_VEL
LIN {X 0,Y 610.24,Z 909.039,A -85,B 0,C 180,E1 866.955,E2 866.955} C_VEL
LIN {X 0,Y 610.173,Z 929.796,A -85,B 0,C 180,E1 869.088,E2 869.088} C_VEL
LIN {X 0,Y 610.115,Z 945.539,A -85,B 0,C 180,E1 871.498,E2 871.498} C_VEL
LIN {X 0,Y 610.098,Z 955.359,A -85,B 0,C 180,E1 873.897,E2 873.897} C_VEL
LIN {X 0,Y 610.105,Z 960.89,A -85,B 0,C 180,E1 876.665,E2 876.665} C_VEL
LIN {X 0,Y 610.171,Z 961.454,A -85,B 0,C 180,E1 878.178,E2 878.178} C_VEL
LIN {X 0,Y 610.156,Z 959.022,A -85,B 0,C 180,E1 880.552,E2 880.552} C_VEL
LIN {X 0,Y 610.142,Z 951.653,A -85,B 0,C 180,E1 883.074,E2 883.074} C_VEL
LIN {X 0,Y 610.151,Z 938.241,A -85,B 0,C 180,E1 885.657,E2 885.657} C_VEL
LIN {X 0,Y 610.234,Z 919.03,A -85,B 0,C 180,E1 888.031,E2 888.031} C_VEL
LIN {X 0,Y 610.287,Z 896.216,A -85,B 0,C 180,E1 889.932,E2 889.932} C_VEL
LIN {X 0,Y 610.363,Z 869.072,A -85,B 0,C 180,E1 891.418,E2 891.418} C_VEL
LIN {X 0,Y 610.17,Z 857.28,A -85,B 0,C 180,E1 891.931,E2 891.931} C_VEL
LIN {X 0,Y 610.06,Z 857.28,A -85,B 0,C 180,E1 892.633,E2 892.633} C_VEL
LIN {X 0,Y 608.734,Z 857.28,A -85,B 0,C 180,E1 893.445,E2 893.445} C_VEL
LIN {X 0,Y 601.931,Z 857.28,A -85,B 0,C 180,E1 895.651,E2 895.651} C_VEL
LIN {X 0,Y 601.813,Z 857.28,A -85,B 0,C 180,E1 895.861,E2 895.861} C_VEL
LIN {X 0,Y 601.892,Z 857.28,A -85,B 0,C 180,E1 900.018,E2 900.018} C_VEL
LIN {X 0,Y 602.003,Z 857.28,A -85,B 0,C 180,E1 904.344,E2 904.344} C_VEL
LIN {X 0,Y 602.014,Z 857.28,A -85,B 0,C 180,E1 908.694,E2 908.694} C_VEL
LIN {X 0,Y 602.063,Z 857.28,A -85,B 0,C 180,E1 913.094,E2 913.094} C_VEL
LIN {X 0,Y 601.865,Z 857.28,A -85,B 0,C 180,E1 919.1,E2 919.1} C_VEL
LIN {X 0,Y 601.78,Z 857.28,A -85,B 0,C 180,E1 923.748,E2 923.748} C_VEL
LIN {X 0,Y 601.787,Z 857.28,A -85,B 0,C 180,E1 928.565,E2 928.565} C_VEL
LIN {X 0,Y 601.837,Z 857.28,A -85,B 0,C 180,E1 933.882,E2 933.882} C_VEL
LIN {X 0,Y 601.778,Z 857.28,A -85,B 0,C 180,E1 938.98,E2 938.98} C_VEL
LIN {X 0,Y 601.74,Z 857.28,A -85,B 0,C 180,E1 945.209,E2 945.209} C_VEL
LIN {X 0,Y 601.735,Z 857.28,A -85,B 0,C 180,E1 951.261,E2 951.261} C_VEL
LIN {X 0,Y 601.529,Z 857.28,A -85,B 0,C 180,E1 956.376,E2 956.376} C_VEL
LIN {X 0,Y 601.688,Z 857.28,A -85,B 0,C 180,E1 961.438,E2 961.438} C_VEL
LIN {X 0,Y 601.954,Z 857.28,A -85,B 0,C 180,E1 966.27,E2 966.27} C_VEL
LIN {X 0,Y 601.73,Z 857.71,A -85,B 0,C 180,E1 967.915,E2 967.915} C_VEL
LIN {X 0,Y 603.05,Z 875.256,A -85,B 0,C 180,E1 968.186,E2 968.186} C_VEL
LIN {X 0,Y 603.145,Z 939.569,A -85,B 0,C 180,E1 969.111,E2 969.111} C_VEL
LIN {X 0,Y 602.964,Z 973.014,A -85,B 0,C 180,E1 970.161,E2 970.161} C_VEL
LIN {X 0,Y 602.788,Z 1005.647,A -85,B 0,C 180,E1 971.796,E2 971.796} C_VEL
LIN {X 0,Y 602.597,Z 1035.507,A -85,B 0,C 180,E1 973.956,E2 973.956} C_VEL
LIN {X 0,Y 602.426,Z 1061.284,A -85,B 0,C 180,E1 976.557,E2 976.557} C_VEL
LIN {X 0,Y 602.305,Z 1080.571,A -85,B 0,C 180,E1 979.23,E2 979.23} C_VEL
LIN {X 0,Y 602.225,Z 1096.654,A -85,B 0,C 180,E1 982.416,E2 982.416} C_VEL
LIN {X 0,Y 602.234,Z 1106.725,A -85,B 0,C 180,E1 985.675,E2 985.675} C_VEL
LIN {X 0,Y 602.185,Z 1110.931,A -85,B 0,C 180,E1 988.56,E2 988.56} C_VEL
LIN {X 0,Y 602.191,Z 1110.93,A -85,B 0,C 180,E1 991.441,E2 991.441} C_VEL
LIN {X 0,Y 602.195,Z 1106.723,A -85,B 0,C 180,E1 994.326,E2 994.326} C_VEL
LIN {X 0,Y 602.19,Z 1096.649,A -85,B 0,C 180,E1 997.586,E2 997.586} C_VEL
LIN {X 0,Y 602.275,Z 1080.586,A -85,B 0,C 180,E1 1000.768,E2 1000.768} C_VEL
LIN {X 0,Y 602.409,Z 1059.67,A -85,B 0,C 180,E1 1003.629,E2 1003.629} C_VEL
LIN {X 0,Y 602.6,Z 1033.536,A -85,B 0,C 180,E1 1006.207,E2 1006.207} C_VEL
LIN {X 0,Y 602.757,Z 1004.104,A -85,B 0,C 180,E1 1008.3,E2 1008.3} C_VEL
LIN {X 0,Y 602.976,Z 971.554,A -85,B 0,C 180,E1 1009.896,E2 1009.896} C_VEL
LIN {X 0,Y 603.083,Z 937.338,A -85,B 0,C 180,E1 1010.944,E2 1010.944} C_VEL
LIN {X 0,Y 602.399,Z 861.939,A -85,B 0,C 180,E1 1012.006,E2 1012.006} C_VEL
LIN {X 0,Y 601.648,Z 857.28,A -85,B 0,C 180,E1 1012.178,E2 1012.178} C_VEL
LIN {X 0,Y 601.872,Z 857.28,A -85,B 0,C 180,E1 1018.309,E2 1018.309} C_VEL
LIN {X 0,Y 601.829,Z 857.28,A -85,B 0,C 180,E1 1023.883,E2 1023.883} C_VEL
LIN {X 0,Y 601.774,Z 857.28,A -85,B 0,C 180,E1 1028.978,E2 1028.978} C_VEL
LIN {X 0,Y 601.717,Z 857.28,A -85,B 0,C 180,E1 1035.205,E2 1035.205} C_VEL
LIN {X 0,Y 601.72,Z 857.28,A -85,B 0,C 180,E1 1041.015,E2 1041.015} C_VEL
LIN {X 0,Y 601.569,Z 857.28,A -85,B 0,C 180,E1 1046.158,E2 1046.158} C_VEL
LIN {X 0,Y 601.666,Z 857.28,A -85,B 0,C 180,E1 1051.429,E2 1051.429} C_VEL
LIN {X 0,Y 601.743,Z 857.28,A -85,B 0,C 180,E1 1056.251,E2 1056.251} C_VEL
LIN {X 0,Y 601.942,Z 857.28,A -85,B 0,C 180,E1 1060.903,E2 1060.903} C_VEL
LIN {X 0,Y 601.552,Z 857.28,A -85,B 0,C 180,E1 1065.41,E2 1065.41} C_VEL
LIN {X 0,Y 601.996,Z 857.28,A -85,B 0,C 180,E1 1069.846,E2 1069.846} C_VEL
LIN {X 0,Y 602.205,Z 857.28,A -85,B 0,C 180,E1 1074.212,E2 1074.212} C_VEL
LIN {X 0,Y 601.884,Z 857.28,A -85,B 0,C 180,E1 1079.982,E2 1079.982} C_VEL
LIN {X 0,Y 601.986,Z 857.28,A -85,B 0,C 180,E1 1084.307,E2 1084.307} C_VEL
LIN {X 0,Y 602.027,Z 857.28,A -85,B 0,C 180,E1 1088.657,E2 1088.657} C_VEL
LIN {X 0,Y 602.073,Z 857.28,A -85,B 0,C 180,E1 1093.056,E2 1093.056} C_VEL
LIN {X 0,Y 602.033,Z 857.28,A -85,B 0,C 180,E1 1097.538,E2 1097.538} C_VEL
LIN {X 0,Y 601.765,Z 857.28,A -85,B 0,C 180,E1 1103.708,E2 1103.708} C_VEL
LIN {X 0,Y 601.795,Z 857.28,A -85,B 0,C 180,E1 1108.522,E2 1108.522} C_VEL
LIN {X 0,Y 601.811,Z 857.28,A -85,B 0,C 180,E1 1113.876,E2 1113.876} C_VEL
LIN {X 0,Y 601.773,Z 857.28,A -85,B 0,C 180,E1 1118.933,E2 1118.933} C_VEL
LIN {X 0,Y 601.729,Z 857.28,A -85,B 0,C 180,E1 1125.207,E2 1125.207} C_VEL
LIN {X 0,Y 601.724,Z 857.28,A -85,B 0,C 180,E1 1131.203,E2 1131.203} C_VEL
LIN {X 0,Y 601.628,Z 857.28,A -85,B 0,C 180,E1 1136.381,E2 1136.381} C_VEL
LIN {X 0,Y 602.204,Z 857.518,A -85,B 0,C 180,E1 1138.856,E2 1138.856} C_VEL
LIN {X 0,Y 602.53,Z 884.135,A -85,B 0,C 180,E1 1140.063,E2 1140.063} C_VEL
LIN {X 0,Y 602.459,Z 909.01,A -85,B 0,C 180,E1 1141.809,E2 1141.809} C_VEL
LIN {X 0,Y 602.355,Z 929.247,A -85,B 0,C 180,E1 1143.903,E2 1143.903} C_VEL
LIN {X 0,Y 602.287,Z 944.832,A -85,B 0,C 180,E1 1146.282,E2 1146.282} C_VEL
LIN {X 0,Y 602.277,Z 955.451,A -85,B 0,C 180,E1 1148.873,E2 1148.873} C_VEL
LIN {X 0,Y 602.223,Z 960.018,A -85,B 0,C 180,E1 1150.922,E2 1150.922} C_VEL
LIN {X 0,Y 602.197,Z 961.445,A -85,B 0,C 180,E1 1152.685,E2 1152.685} C_VEL
LIN {X 0,Y 602.227,Z 959.276,A -85,B 0,C 180,E1 1155.438,E2 1155.438} C_VEL
LIN {X 0,Y 602.222,Z 952.071,A -85,B 0,C 180,E1 1158.028,E2 1158.028} C_VEL
LIN {X 0,Y 602.306,Z 939.288,A -85,B 0,C 180,E1 1160.595,E2 1160.595} C_VEL
LIN {X 0,Y 602.381,Z 920.801,A -85,B 0,C 180,E1 1162.978,E2 1162.978} C_VEL
LIN {X 0,Y 602.531,Z 898.114,A -85,B 0,C 180,E1 1164.954,E2 1164.954} C_VEL
LIN {X 0,Y 602.66,Z 871.466,A -85,B 0,C 180,E1 1166.489,E2 1166.489} C_VEL
LIN {X 0,Y 602.217,Z 857.28,A -85,B 0,C 180,E1 1167.117,E2 1167.117} C_VEL
LIN {X 0,Y 601.975,Z 857.28,A -85,B 0,C 180,E1 1174.327,E2 1174.327} C_VEL
LIN {X 0,Y 602.022,Z 857.28,A -85,B 0,C 180,E1 1178.679,E2 1178.679} C_VEL
LIN {X 0,Y 602.103,Z 857.28,A -85,B 0,C 180,E1 1183.08,E2 1183.08} C_VEL
LIN {X 0,Y 601.995,Z 857.28,A -85,B 0,C 180,E1 1187.566,E2 1187.566} C_VEL
LIN {X 0,Y 601.74,Z 857.28,A -85,B 0,C 180,E1 1193.739,E2 1193.739} C_VEL
LIN {X 0,Y 601.764,Z 857.28,A -85,B 0,C 180,E1 1198.558,E2 1198.558} C_VEL
LIN {X 0,Y 601.825,Z 857.28,A -85,B 0,C 180,E1 1203.949,E2 1203.949} C_VEL
LIN {X 0,Y 601.717,Z 857.28,A -85,B 0,C 180,E1 1208.981,E2 1208.981} C_VEL
LIN {X 0,Y 601.731,Z 857.28,A -85,B 0,C 180,E1 1215.258,E2 1215.258} C_VEL
LIN {X 0,Y 601.686,Z 857.28,A -85,B 0,C 180,E1 1219.182,E2 1219.182} C_VEL
LIN {X 0,Y 601.844,Z 857.551,A -85,B 0,C 180,E1 1223.849,E2 1223.849} C_VEL
LIN {X 0,Y 602.564,Z 884.442,A -85,B 0,C 180,E1 1225.081,E2 1225.081} C_VEL
LIN {X 0,Y 602.435,Z 908.916,A -85,B 0,C 180,E1 1226.8,E2 1226.8} C_VEL
LIN {X 0,Y 602.329,Z 930.042,A -85,B 0,C 180,E1 1229.001,E2 1229.001} C_VEL
LIN {X 0,Y 602.227,Z 945.984,A -85,B 0,C 180,E1 1231.5,E2 1231.5} C_VEL
LIN {X 0,Y 602.219,Z 955.633,A -85,B 0,C 180,E1 1233.93,E2 1233.93} C_VEL
LIN {X 0,Y 602.215,Z 960.504,A -85,B 0,C 180,E1 1236.311,E2 1236.311} C_VEL
LIN {X 0,Y 602.241,Z 961.389,A -85,B 0,C 180,E1 1238.466,E2 1238.466} C_VEL
LIN {X 0,Y 602.251,Z 958.247,A -85,B 0,C 180,E1 1240.952,E2 1240.952} C_VEL
LIN {X 0,Y 602.271,Z 949.384,A -85,B 0,C 180,E1 1243.685,E2 1243.685} C_VEL
LIN {X 0,Y 602.315,Z 935.237,A -85,B 0,C 180,E1 1246.209,E2 1246.209} C_VEL
LIN {X 0,Y 602.406,Z 916.42,A -85,B 0,C 180,E1 1248.424,E2 1248.424} C_VEL
LIN {X 0,Y 602.509,Z 892.344,A -85,B 0,C 180,E1 1250.348,E2 1250.348} C_VEL
LIN {X 0,Y 602.665,Z 865.092,A -85,B 0,C 180,E1 1251.762,E2 1251.762} C_VEL
LIN {X 0,Y 602.251,Z 857.28,A -85,B 0,C 180,E1 1252.074,E2 1252.074} C_VEL
LIN {X 0,Y 601.813,Z 857.28,A -85,B 0,C 180,E1 1255.861,E2 1255.861} C_VEL
LIN {X 0,Y 597.989,Z 857.28,A -85,B 0,C 180,E1 1257.486,E2 1257.486} C_VEL
LIN {X 0,Y 594.093,Z 857.28,A -85,B 0,C 180,E1 1259.132,E2 1259.132} C_VEL
LIN {X 0,Y 594.085,Z 857.28,A -85,B 0,C 180,E1 1264.402,E2 1264.402} C_VEL
LIN {X 0,Y 594.094,Z 857.28,A -85,B 0,C 180,E1 1268.811,E2 1268.811} C_VEL
LIN {X 0,Y 593.851,Z 857.28,A -85,B 0,C 180,E1 1274.342,E2 1274.342} C_VEL
LIN {X 0,Y 593.904,Z 857.28,A -85,B 0,C 180,E1 1279.394,E2 1279.394} C_VEL
LIN {X 0,Y 593.857,Z 857.28,A -85,B 0,C 180,E1 1284.084,E2 1284.084} C_VEL
LIN {X 0,Y 593.776,Z 857.28,A -85,B 0,C 180,E1 1288.986,E2 1288.986} C_VEL
LIN {X 0,Y 593.895,Z 857.28,A -85,B 0,C 180,E1 1294.122,E2 1294.122} C_VEL
LIN {X 0,Y 593.693,Z 857.28,A -85,B 0,C 180,E1 1300.087,E2 1300.087} C_VEL
LIN {X 0,Y 593.806,Z 857.28,A -85,B 0,C 180,E1 1305.558,E2 1305.558} C_VEL
LIN {X 0,Y 593.74,Z 857.28,A -85,B 0,C 180,E1 1310.394,E2 1310.394} C_VEL
LIN {X 0,Y 593.663,Z 857.28,A -85,B 0,C 180,E1 1315.87,E2 1315.87} C_VEL
LIN {X 0,Y 593.776,Z 857.28,A -85,B 0,C 180,E1 1321.022,E2 1321.022} C_VEL
LIN {X 0,Y 594,Z 857.28,A -85,B 0,C 180,E1 1326.571,E2 1326.571} C_VEL
LIN {X 0,Y 593.837,Z 857.293,A -85,B 0,C 180,E1 1327.6,E2 1327.6} C_VEL
LIN {X 0,Y 595.701,Z 869.591,A -85,B 0,C 180,E1 1327.831,E2 1327.831} C_VEL
LIN {X 0,Y 595.763,Z 939.568,A -85,B 0,C 180,E1 1328.84,E2 1328.84} C_VEL
LIN {X 0,Y 595.49,Z 973.452,A -85,B 0,C 180,E1 1329.919,E2 1329.919} C_VEL
LIN {X 0,Y 595.193,Z 1005.649,A -85,B 0,C 180,E1 1331.556,E2 1331.556} C_VEL
LIN {X 0,Y 594.883,Z 1035.507,A -85,B 0,C 180,E1 1333.742,E2 1333.742} C_VEL
LIN {X 0,Y 594.639,Z 1061.431,A -85,B 0,C 180,E1 1336.395,E2 1336.395} C_VEL
LIN {X 0,Y 594.442,Z 1081.021,A -85,B 0,C 180,E1 1339.162,E2 1339.162} C_VEL
LIN {X 0,Y 594.344,Z 1096.653,A -85,B 0,C 180,E1 1342.315,E2 1342.315} C_VEL
LIN {X 0,Y 594.33,Z 1106.726,A -85,B 0,C 180,E1 1345.617,E2 1345.617} C_VEL
LIN {X 0,Y 594.281,Z 1110.931,A -85,B 0,C 180,E1 1348.541,E2 1348.541} C_VEL
LIN {X 0,Y 594.288,Z 1110.931,A -85,B 0,C 180,E1 1351.46,E2 1351.46} C_VEL
LIN {X 0,Y 594.294,Z 1106.723,A -85,B 0,C 180,E1 1354.384,E2 1354.384} C_VEL
LIN {X 0,Y 594.309,Z 1096.649,A -85,B 0,C 180,E1 1357.687,E2 1357.687} C_VEL
LIN {X 0,Y 594.414,Z 1081.051,A -85,B 0,C 180,E1 1360.833,E2 1360.833} C_VEL
LIN {X 0,Y 594.635,Z 1059.913,A -85,B 0,C 180,E1 1363.783,E2 1363.783} C_VEL
LIN {X 0,Y 594.906,Z 1033.789,A -85,B 0,C 180,E1 1366.402,E2 1366.402} C_VEL
LIN {X 0,Y 595.191,Z 1004.102,A -85,B 0,C 180,E1 1368.541,E2 1368.541} C_VEL
LIN {X 0,Y 595.476,Z 971.516,A -85,B 0,C 180,E1 1370.159,E2 1370.159} C_VEL
LIN {X 0,Y 595.691,Z 937.338,A -85,B 0,C 180,E1 1371.216,E2 1371.216} C_VEL
LIN {X 0,Y 594.967,Z 862.607,A -85,B 0,C 180,E1 1372.287,E2 1372.287} C_VEL
LIN {X 0,Y 593.746,Z 857.28,A -85,B 0,C 180,E1 1372.49,E2 1372.49} C_VEL
LIN {X 0,Y 593.896,Z 857.28,A -85,B 0,C 180,E1 1377.316,E2 1377.316} C_VEL
LIN {X 0,Y 593.859,Z 857.28,A -85,B 0,C 180,E1 1382.721,E2 1382.721} C_VEL
LIN {X 0,Y 593.732,Z 857.28,A -85,B 0,C 180,E1 1387.766,E2 1387.766} C_VEL
LIN {X 0,Y 593.697,Z 857.28,A -85,B 0,C 180,E1 1393.518,E2 1393.518} C_VEL
LIN {X 0,Y 593.788,Z 857.28,A -85,B 0,C 180,E1 1398.471,E2 1398.471} C_VEL
LIN {X 0,Y 593.855,Z 857.28,A -85,B 0,C 180,E1 1404.093,E2 1404.093} C_VEL
LIN {X 0,Y 593.841,Z 857.28,A -85,B 0,C 180,E1 1410.099,E2 1410.099} C_VEL
LIN {X 0,Y 593.915,Z 857.28,A -85,B 0,C 180,E1 1415.918,E2 1415.918} C_VEL
LIN {X 0,Y 594.021,Z 857.28,A -85,B 0,C 180,E1 1420.638,E2 1420.638} C_VEL
LIN {X 0,Y 593.712,Z 857.28,A -85,B 0,C 180,E1 1425.213,E2 1425.213} C_VEL
LIN {X 0,Y 594.055,Z 857.28,A -85,B 0,C 180,E1 1429.708,E2 1429.708} C_VEL
LIN {X 0,Y 594.267,Z 857.28,A -85,B 0,C 180,E1 1434.134,E2 1434.134} C_VEL
LIN {X 0,Y 593.984,Z 857.28,A -85,B 0,C 180,E1 1439.981,E2 1439.981} C_VEL
LIN {X 0,Y 594.069,Z 857.28,A -85,B 0,C 180,E1 1444.364,E2 1444.364} C_VEL
LIN {X 0,Y 594.102,Z 857.28,A -85,B 0,C 180,E1 1448.773,E2 1448.773} C_VEL
LIN {X 0,Y 593.861,Z 857.28,A -85,B 0,C 180,E1 1454.341,E2 1454.341} C_VEL
LIN {X 0,Y 593.912,Z 857.28,A -85,B 0,C 180,E1 1459.393,E2 1459.393} C_VEL
LIN {X 0,Y 593.835,Z 857.28,A -85,B 0,C 180,E1 1464.044,E2 1464.044} C_VEL
LIN {X 0,Y 593.784,Z 857.28,A -85,B 0,C 180,E1 1468.943,E2 1468.943} C_VEL
LIN {X 0,Y 593.875,Z 857.28,A -85,B 0,C 180,E1 1474.078,E2 1474.078} C_VEL
LIN {X 0,Y 593.676,Z 857.28,A -85,B 0,C 180,E1 1480.083,E2 1480.083} C_VEL
LIN {X 0,Y 593.833,Z 857.28,A -85,B 0,C 180,E1 1485.502,E2 1485.502} C_VEL
LIN {X 0,Y 593.728,Z 857.28,A -85,B 0,C 180,E1 1490.391,E2 1490.391} C_VEL
LIN {X 0,Y 593.77,Z 857.28,A -85,B 0,C 180,E1 1495.875,E2 1495.875} C_VEL
LIN {X 0,Y 594.288,Z 858.017,A -85,B 0,C 180,E1 1498.681,E2 1498.681} C_VEL
LIN {X 0,Y 594.79,Z 884.981,A -85,B 0,C 180,E1 1499.94,E2 1499.94} C_VEL
LIN {X 0,Y 594.647,Z 910.144,A -85,B 0,C 180,E1 1501.762,E2 1501.762} C_VEL
LIN {X 0,Y 594.486,Z 930.938,A -85,B 0,C 180,E1 1503.996,E2 1503.996} C_VEL
LIN {X 0,Y 594.406,Z 945.847,A -85,B 0,C 180,E1 1506.387,E2 1506.387} C_VEL
LIN {X 0,Y 594.356,Z 956.272,A -85,B 0,C 180,E1 1509.105,E2 1509.105} C_VEL
LIN {X 0,Y 594.296,Z 959.634,A -85,B 0,C 180,E1 1510.658,E2 1510.658} C_VEL
LIN {X 0,Y 594.259,Z 961.288,A -85,B 0,C 180,E1 1512.197,E2 1512.197} C_VEL
LIN {X 0,Y 594.264,Z 961.281,A -85,B 0,C 180,E1 1513.724,E2 1513.724} C_VEL
LIN {X 0,Y 594.335,Z 958.161,A -85,B 0,C 180,E1 1516.033,E2 1516.033} C_VEL
LIN {X 0,Y 594.353,Z 949.797,A -85,B 0,C 180,E1 1518.662,E2 1518.662} C_VEL
LIN {X 0,Y 594.454,Z 935.966,A -85,B 0,C 180,E1 1521.209,E2 1521.209} C_VEL
LIN {X 0,Y 594.581,Z 916.701,A -85,B 0,C 180,E1 1523.536,E2 1523.536} C_VEL
LIN {X 0,Y 594.768,Z 893.454,A -85,B 0,C 180,E1 1525.437,E2 1525.437} C_VEL
LIN {X 0,Y 594.996,Z 866.169,A -85,B 0,C 180,E1 1526.9,E2 1526.9} C_VEL
LIN {X 0,Y 594.248,Z 857.28,A -85,B 0,C 180,E1 1527.261,E2 1527.261} C_VEL
LIN {X 0,Y 594.059,Z 857.28,A -85,B 0,C 180,E1 1534.385,E2 1534.385} C_VEL
LIN {X 0,Y 594.086,Z 857.28,A -85,B 0,C 180,E1 1538.795,E2 1538.795} C_VEL
LIN {X 0,Y 593.844,Z 857.28,A -85,B 0,C 180,E1 1544.509,E2 1544.509} C_VEL
LIN {X 0,Y 593.867,Z 857.28,A -85,B 0,C 180,E1 1549.509,E2 1549.509} C_VEL
LIN {X 0,Y 593.808,Z 857.28,A -85,B 0,C 180,E1 1554.076,E2 1554.076} C_VEL
LIN {X 0,Y 593.755,Z 857.28,A -85,B 0,C 180,E1 1558.979,E2 1558.979} C_VEL
LIN {X 0,Y 593.886,Z 857.28,A -85,B 0,C 180,E1 1564.116,E2 1564.116} C_VEL
LIN {X 0,Y 593.631,Z 857.28,A -85,B 0,C 180,E1 1570.137,E2 1570.137} C_VEL
LIN {X 0,Y 593.839,Z 857.28,A -85,B 0,C 180,E1 1575.552,E2 1575.552} C_VEL
LIN {X 0,Y 593.66,Z 857.28,A -85,B 0,C 180,E1 1580.431,E2 1580.431} C_VEL
LIN {X 0,Y 593.922,Z 857.732,A -85,B 0,C 180,E1 1583.662,E2 1583.662} C_VEL
LIN {X 0,Y 594.827,Z 883.212,A -85,B 0,C 180,E1 1584.842,E2 1584.842} C_VEL
LIN {X 0,Y 594.627,Z 908.436,A -85,B 0,C 180,E1 1586.609,E2 1586.609} C_VEL
LIN {X 0,Y 594.497,Z 929.96,A -85,B 0,C 180,E1 1588.871,E2 1588.871} C_VEL
LIN {X 0,Y 594.37,Z 945.324,A -85,B 0,C 180,E1 1591.285,E2 1591.285} C_VEL
LIN {X 0,Y 594.367,Z 955.153,A -85,B 0,C 180,E1 1593.722,E2 1593.722} C_VEL
LIN {X 0,Y 594.295,Z 960.763,A -85,B 0,C 180,E1 1596.514,E2 1596.514} C_VEL
LIN {X 0,Y 594.322,Z 960.999,A -85,B 0,C 180,E1 1599.134,E2 1599.134} C_VEL
LIN {X 0,Y 594.331,Z 956.173,A -85,B 0,C 180,E1 1601.844,E2 1601.844} C_VEL
LIN {X 0,Y 594.435,Z 945.886,A -85,B 0,C 180,E1 1604.514,E2 1604.514} C_VEL
LIN {X 0,Y 594.488,Z 930.57,A -85,B 0,C 180,E1 1606.961,E2 1606.961} C_VEL
LIN {X 0,Y 594.685,Z 909.921,A -85,B 0,C 180,E1 1609.168,E2 1609.168} C_VEL
LIN {X 0,Y 594.863,Z 885.078,A -85,B 0,C 180,E1 1610.962,E2 1610.962} C_VEL
LIN {X 0,Y 594.332,Z 857.28,A -85,B 0,C 180,E1 1612.291,E2 1612.291} C_VEL
LIN {X 0,Y 594.235,Z 857.28,A -85,B 0,C 180,E1 1618.559,E2 1618.559} C_VEL
LIN {X 0,Y 594.093,Z 857.28,A -85,B 0,C 180,E1 1619.132,E2 1619.132} C_VEL
LIN {X 0,Y 589.938,Z 857.28,A -85,B 0,C 180,E1 1620.775,E2 1620.775} C_VEL
LIN {X 0,Y 586.107,Z 857.28,A -85,B 0,C 180,E1 1622.441,E2 1622.441} C_VEL
LIN {X 0,Y 586.12,Z 857.28,A -85,B 0,C 180,E1 1627.437,E2 1627.437} C_VEL
LIN {X 0,Y 586.151,Z 857.28,A -85,B 0,C 180,E1 1633.457,E2 1633.457} C_VEL
LIN {X 0,Y 585.994,Z 857.28,A -85,B 0,C 180,E1 1639.638,E2 1639.638} C_VEL
LIN {X 0,Y 585.894,Z 857.28,A -85,B 0,C 180,E1 1644.433,E2 1644.433} C_VEL
LIN {X 0,Y 585.798,Z 857.28,A -85,B 0,C 180,E1 1649.419,E2 1649.419} C_VEL
LIN {X 0,Y 585.885,Z 857.28,A -85,B 0,C 180,E1 1654.654,E2 1654.654} C_VEL
LIN {X 0,Y 585.778,Z 857.28,A -85,B 0,C 180,E1 1660.258,E2 1660.258} C_VEL
LIN {X 0,Y 585.931,Z 857.28,A -85,B 0,C 180,E1 1666.348,E2 1666.348} C_VEL
LIN {X 0,Y 585.841,Z 857.28,A -85,B 0,C 180,E1 1671.665,E2 1671.665} C_VEL
LIN {X 0,Y 585.74,Z 857.28,A -85,B 0,C 180,E1 1677.124,E2 1677.124} C_VEL
LIN {X 0,Y 585.811,Z 857.28,A -85,B 0,C 180,E1 1682.276,E2 1682.276} C_VEL
LIN {X 0,Y 585.965,Z 857.28,A -85,B 0,C 180,E1 1687.269,E2 1687.269} C_VEL
LIN {X 0,Y 588.411,Z 870.965,A -85,B 0,C 180,E1 1687.559,E2 1687.559} C_VEL
LIN {X 0,Y 588.406,Z 939.351,A -85,B 0,C 180,E1 1688.557,E2 1688.557} C_VEL
LIN {X 0,Y 588.057,Z 972.002,A -85,B 0,C 180,E1 1689.595,E2 1689.595} C_VEL
LIN {X 0,Y 587.653,Z 1004.117,A -85,B 0,C 180,E1 1691.213,E2 1691.213} C_VEL
LIN {X 0,Y 587.202,Z 1033.997,A -85,B 0,C 180,E1 1693.394,E2 1693.394} C_VEL
LIN {X 0,Y 586.859,Z 1059.039,A -85,B 0,C 180,E1 1695.927,E2 1695.927} C_VEL
LIN {X 0,Y 586.624,Z 1080.208,A -85,B 0,C 180,E1 1698.875,E2 1698.875} C_VEL
LIN {X 0,Y 586.469,Z 1096.653,A -85,B 0,C 180,E1 1702.211,E2 1702.211} C_VEL
LIN {X 0,Y 586.429,Z 1106.726,A -85,B 0,C 180,E1 1705.558,E2 1705.558} C_VEL
LIN {X 0,Y 586.378,Z 1110.932,A -85,B 0,C 180,E1 1708.521,E2 1708.521} C_VEL
LIN {X 0,Y 586.385,Z 1110.931,A -85,B 0,C 180,E1 1711.48,E2 1711.48} C_VEL
LIN {X 0,Y 586.395,Z 1106.724,A -85,B 0,C 180,E1 1714.443,E2 1714.443} C_VEL
LIN {X 0,Y 586.439,Z 1096.649,A -85,B 0,C 180,E1 1717.791,E2 1717.791} C_VEL
LIN {X 0,Y 586.607,Z 1080.259,A -85,B 0,C 180,E1 1721.116,E2 1721.116} C_VEL
LIN {X 0,Y 586.853,Z 1059.027,A -85,B 0,C 180,E1 1724.074,E2 1724.074} C_VEL
LIN {X 0,Y 587.2,Z 1033.984,A -85,B 0,C 180,E1 1726.607,E2 1726.607} C_VEL
LIN {X 0,Y 587.624,Z 1004.099,A -85,B 0,C 180,E1 1728.789,E2 1728.789} C_VEL
LIN {X 0,Y 588.015,Z 971.711,A -85,B 0,C 180,E1 1730.419,E2 1730.419} C_VEL
LIN {X 0,Y 588.341,Z 937.508,A -85,B 0,C 180,E1 1731.491,E2 1731.491} C_VEL
LIN {X 0,Y 587.847,Z 864.647,A -85,B 0,C 180,E1 1732.546,E2 1732.546} C_VEL
LIN {X 0,Y 585.89,Z 857.28,A -85,B 0,C 180,E1 1732.808,E2 1732.808} C_VEL
LIN {X 0,Y 585.856,Z 857.28,A -85,B 0,C 180,E1 1738.521,E2 1738.521} C_VEL
LIN {X 0,Y 585.873,Z 857.28,A -85,B 0,C 180,E1 1744.65,E2 1744.65} C_VEL
LIN {X 0,Y 585.8,Z 857.28,A -85,B 0,C 180,E1 1750.253,E2 1750.253} C_VEL
LIN {X 0,Y 585.926,Z 857.28,A -85,B 0,C 180,E1 1756.348,E2 1756.348} C_VEL
LIN {X 0,Y 585.867,Z 857.28,A -85,B 0,C 180,E1 1761.662,E2 1761.662} C_VEL
LIN {X 0,Y 585.742,Z 857.28,A -85,B 0,C 180,E1 1767.117,E2 1767.117} C_VEL
LIN {X 0,Y 585.795,Z 857.28,A -85,B 0,C 180,E1 1772.266,E2 1772.266} C_VEL
LIN {X 0,Y 585.872,Z 857.28,A -85,B 0,C 180,E1 1777.182,E2 1777.182} C_VEL
LIN {X 0,Y 586.097,Z 857.28,A -85,B 0,C 180,E1 1781.929,E2 1781.929} C_VEL
LIN {X 0,Y 585.82,Z 857.28,A -85,B 0,C 180,E1 1788.053,E2 1788.053} C_VEL
LIN {X 0,Y 586.345,Z 857.28,A -85,B 0,C 180,E1 1794.055,E2 1794.055} C_VEL
LIN {X 0,Y 586.094,Z 857.28,A -85,B 0,C 180,E1 1799.981,E2 1799.981} C_VEL
LIN {X 0,Y 586.158,Z 857.28,A -85,B 0,C 180,E1 1804.423,E2 1804.423} C_VEL
LIN {X 0,Y 586.163,Z 857.28,A -85,B 0,C 180,E1 1808.893,E2 1808.893} C_VEL
LIN {X 0,Y 586.161,Z 857.28,A -85,B 0,C 180,E1 1813.417,E2 1813.417} C_VEL
LIN {X 0,Y 586.002,Z 857.28,A -85,B 0,C 180,E1 1819.597,E2 1819.597} C_VEL
LIN {X 0,Y 585.842,Z 857.28,A -85,B 0,C 180,E1 1825.235,E2 1825.235} C_VEL
LIN {X 0,Y 585.807,Z 857.28,A -85,B 0,C 180,E1 1829.375,E2 1829.375} C_VEL
LIN {X 0,Y 585.881,Z 857.28,A -85,B 0,C 180,E1 1834.608,E2 1834.608} C_VEL
LIN {X 0,Y 585.778,Z 857.28,A -85,B 0,C 180,E1 1840.209,E2 1840.209} C_VEL
LIN {X 0,Y 585.912,Z 857.28,A -85,B 0,C 180,E1 1846.296,E2 1846.296} C_VEL
LIN {X 0,Y 585.831,Z 857.28,A -85,B 0,C 180,E1 1851.663,E2 1851.663} C_VEL
LIN {X 0,Y 585.907,Z 857.28,A -85,B 0,C 180,E1 1857.134,E2 1857.134} C_VEL
LIN {X 0,Y 586.25,Z 857.28,A -85,B 0,C 180,E1 1858.441,E2 1858.441} C_VEL
LIN {X 0,Y 587.117,Z 883.809,A -85,B 0,C 180,E1 1859.7,E2 1859.7} C_VEL
LIN {X 0,Y 586.881,Z 908.877,A -85,B 0,C 180,E1 1861.497,E2 1861.497} C_VEL
LIN {X 0,Y 586.629,Z 930.411,A -85,B 0,C 180,E1 1863.808,E2 1863.808} C_VEL
LIN {X 0,Y 586.534,Z 946.312,A -85,B 0,C 180,E1 1866.397,E2 1866.397} C_VEL
LIN {X 0,Y 586.47,Z 956.669,A -85,B 0,C 180,E1 1869.207,E2 1869.207} C_VEL
LIN {X 0,Y 586.352,Z 961.127,A -85,B 0,C 180,E1 1871.948,E2 1871.948} C_VEL
LIN {X 0,Y 586.338,Z 961.384,A -85,B 0,C 180,E1 1873.497,E2 1873.497} C_VEL
LIN {X 0,Y 586.425,Z 958.549,A -85,B 0,C 180,E1 1875.889,E2 1875.889} C_VEL
LIN {X 0,Y 586.483,Z 949.804,A -85,B 0,C 180,E1 1878.737,E2 1878.737} C_VEL
LIN {X 0,Y 586.59,Z 936.246,A -85,B 0,C 180,E1 1881.277,E2 1881.277} C_VEL
LIN {X 0,Y 586.762,Z 917.559,A -85,B 0,C 180,E1 1883.594,E2 1883.594} C_VEL
LIN {X 0,Y 587.02,Z 894.075,A -85,B 0,C 180,E1 1885.562,E2 1885.562} C_VEL
LIN {X 0,Y 587.307,Z 867.118,A -85,B 0,C 180,E1 1887.044,E2 1887.044} C_VEL
LIN {X 0,Y 586.249,Z 857.28,A -85,B 0,C 180,E1 1887.502,E2 1887.502} C_VEL
LIN {X 0,Y 586.144,Z 857.28,A -85,B 0,C 180,E1 1894.444,E2 1894.444} C_VEL
LIN {X 0,Y 586.148,Z 857.28,A -85,B 0,C 180,E1 1898.915,E2 1898.915} C_VEL
LIN {X 0,Y 586.193,Z 857.28,A -85,B 0,C 180,E1 1903.441,E2 1903.441} C_VEL
LIN {X 0,Y 585.963,Z 857.28,A -85,B 0,C 180,E1 1909.627,E2 1909.627} C_VEL
LIN {X 0,Y 585.849,Z 857.28,A -85,B 0,C 180,E1 1914.425,E2 1914.425} C_VEL
LIN {X 0,Y 585.784,Z 857.28,A -85,B 0,C 180,E1 1919.412,E2 1919.412} C_VEL
LIN {X 0,Y 585.894,Z 857.28,A -85,B 0,C 180,E1 1924.647,E2 1924.647} C_VEL
LIN {X 0,Y 585.733,Z 857.28,A -85,B 0,C 180,E1 1930.257,E2 1930.257} C_VEL
LIN {X 0,Y 585.931,Z 857.28,A -85,B 0,C 180,E1 1936.346,E2 1936.346} C_VEL
LIN {X 0,Y 585.739,Z 857.28,A -85,B 0,C 180,E1 1941.7,E2 1941.7} C_VEL
LIN {X 0,Y 585.962,Z 857.28,A -85,B 0,C 180,E1 1943.436,E2 1943.436} C_VEL
LIN {X 0,Y 587.135,Z 879.064,A -85,B 0,C 180,E1 1944.436,E2 1944.436} C_VEL
LIN {X 0,Y 586.883,Z 904.828,A -85,B 0,C 180,E1 1946.154,E2 1946.154} C_VEL
LIN {X 0,Y 586.664,Z 925.18,A -85,B 0,C 180,E1 1948.155,E2 1948.155} C_VEL
LIN {X 0,Y 586.533,Z 942.516,A -85,B 0,C 180,E1 1950.664,E2 1950.664} C_VEL
LIN {X 0,Y 586.472,Z 954.257,A -85,B 0,C 180,E1 1953.372,E2 1953.372} C_VEL
LIN {X 0,Y 586.431,Z 959.643,A -85,B 0,C 180,E1 1955.633,E2 1955.633} C_VEL
LIN {X 0,Y 586.358,Z 961.414,A -85,B 0,C 180,E1 1958.368,E2 1958.368} C_VEL
LIN {X 0,Y 586.454,Z 957.899,A -85,B 0,C 180,E1 1961.201,E2 1961.201} C_VEL
LIN {X 0,Y 586.539,Z 949.07,A -85,B 0,C 180,E1 1963.916,E2 1963.916} C_VEL
LIN {X 0,Y 586.595,Z 934.122,A -85,B 0,C 180,E1 1966.593,E2 1966.593} C_VEL
LIN {X 0,Y 586.767,Z 915.149,A -85,B 0,C 180,E1 1968.833,E2 1968.833} C_VEL
LIN {X 0,Y 587.005,Z 891.36,A -85,B 0,C 180,E1 1970.746,E2 1970.746} C_VEL
LIN {X 0,Y 587.298,Z 864.593,A -85,B 0,C 180,E1 1972.151,E2 1972.151} C_VEL
LIN {X 0,Y 586.404,Z 857.28,A -85,B 0,C 180,E1 1972.512,E2 1972.512} C_VEL
LIN {X 0,Y 586.194,Z 857.28,A -85,B 0,C 180,E1 1979.118,E2 1979.118} C_VEL
LIN {X 0,Y 586.107,Z 857.28,A -85,B 0,C 180,E1 1982.441,E2 1982.441} C_VEL
LIN {X 0,Y 583.686,Z 857.28,A -85,B 0,C 180,E1 1983.704,E2 1983.704} C_VEL
LIN {X 0,Y 578.219,Z 857.28,A -85,B 0,C 180,E1 1985.595,E2 1985.595} C_VEL
LIN {X 0,Y 578.112,Z 857.28,A -85,B 0,C 180,E1 1985.814,E2 1985.814} C_VEL
LIN {X 0,Y 578.016,Z 857.28,A -85,B 0,C 180,E1 1990.58,E2 1990.58} C_VEL
LIN {X 0,Y 577.958,Z 857.28,A -85,B 0,C 180,E1 1995.2,E2 1995.2} C_VEL
LIN {X 0,Y 578.068,Z 857.28,A -85,B 0,C 180,E1 1999.919,E2 1999.919} C_VEL
LIN {X 0,Y 577.988,Z 857.28,A -85,B 0,C 180,E1 2004.789,E2 2004.789} C_VEL
LIN {X 0,Y 577.83,Z 857.28,A -85,B 0,C 180,E1 2010.153,E2 2010.153} C_VEL
LIN {X 0,Y 577.865,Z 857.28,A -85,B 0,C 180,E1 2015.206,E2 2015.206} C_VEL
LIN {X 0,Y 577.834,Z 857.28,A -85,B 0,C 180,E1 2020.929,E2 2020.929} C_VEL
LIN {X 0,Y 577.977,Z 857.28,A -85,B 0,C 180,E1 2027.071,E2 2027.071} C_VEL
LIN {X 0,Y 577.956,Z 857.28,A -85,B 0,C 180,E1 2032.949,E2 2032.949} C_VEL
LIN {X 0,Y 577.916,Z 857.28,A -85,B 0,C 180,E1 2038.401,E2 2038.401} C_VEL
LIN {X 0,Y 578.03,Z 857.28,A -85,B 0,C 180,E1 2043.558,E2 2043.558} C_VEL
LIN {X 0,Y 578.098,Z 857.28,A -85,B 0,C 180,E1 2046.944,E2 2046.944} C_VEL
LIN {X 0,Y 581.126,Z 870.854,A -85,B 0,C 180,E1 2047.261,E2 2047.261} C_VEL
LIN {X 0,Y 581.063,Z 939.35,A -85,B 0,C 180,E1 2048.272,E2 2048.272} C_VEL
LIN {X 0,Y 580.586,Z 973.762,A -85,B 0,C 180,E1 2049.393,E2 2049.393} C_VEL
LIN {X 0,Y 580.06,Z 1005.651,A -85,B 0,C 180,E1 2051.057,E2 2051.057} C_VEL
LIN {X 0,Y 579.5,Z 1035.506,A -85,B 0,C 180,E1 2053.298,E2 2053.298} C_VEL
LIN {X 0,Y 579.087,Z 1061.037,A -85,B 0,C 180,E1 2055.975,E2 2055.975} C_VEL
LIN {X 0,Y 578.774,Z 1081.247,A -85,B 0,C 180,E1 2058.904,E2 2058.904} C_VEL
LIN {X 0,Y 578.596,Z 1096.653,A -85,B 0,C 180,E1 2062.104,E2 2062.104} C_VEL
LIN {X 0,Y 578.528,Z 1106.727,A -85,B 0,C 180,E1 2065.497,E2 2065.497} C_VEL
LIN {X 0,Y 578.475,Z 1110.932,A -85,B 0,C 180,E1 2068.501,E2 2068.501} C_VEL
LIN {X 0,Y 578.482,Z 1110.931,A -85,B 0,C 180,E1 2071.5,E2 2071.5} C_VEL
LIN {X 0,Y 578.497,Z 1106.724,A -85,B 0,C 180,E1 2074.504,E2 2074.504} C_VEL
LIN {X 0,Y 578.574,Z 1096.649,A -85,B 0,C 180,E1 2077.897,E2 2077.897} C_VEL
LIN {X 0,Y 578.784,Z 1080.26,A -85,B 0,C 180,E1 2081.268,E2 2081.268} C_VEL
LIN {X 0,Y 579.06,Z 1059.884,A -85,B 0,C 180,E1 2084.164,E2 2084.164} C_VEL
LIN {X 0,Y 579.514,Z 1034.237,A -85,B 0,C 180,E1 2086.812,E2 2086.812} C_VEL
LIN {X 0,Y 580.038,Z 1005.633,A -85,B 0,C 180,E1 2088.945,E2 2088.945} C_VEL
LIN {X 0,Y 580.551,Z 972.942,A -85,B 0,C 180,E1 2090.642,E2 2090.642} C_VEL
LIN {X 0,Y 580.989,Z 937.508,A -85,B 0,C 180,E1 2091.776,E2 2091.776} C_VEL
LIN {X 0,Y 580.52,Z 866.074,A -85,B 0,C 180,E1 2092.827,E2 2092.827} C_VEL
LIN {X 0,Y 577.954,Z 857.28,A -85,B 0,C 180,E1 2093.139,E2 2093.139} C_VEL
LIN {X 0,Y 577.986,Z 857.28,A -85,B 0,C 180,E1 2098.134,E2 2098.134} C_VEL
LIN {X 0,Y 578.035,Z 857.28,A -85,B 0,C 180,E1 2103.372,E2 2103.372} C_VEL
LIN {X 0,Y 577.896,Z 857.28,A -85,B 0,C 180,E1 2108.962,E2 2108.962} C_VEL
LIN {X 0,Y 577.938,Z 857.28,A -85,B 0,C 180,E1 2115.02,E2 2115.02} C_VEL
LIN {X 0,Y 577.939,Z 857.28,A -85,B 0,C 180,E1 2121.038,E2 2121.038} C_VEL
LIN {X 0,Y 577.855,Z 857.28,A -85,B 0,C 180,E1 2126.978,E2 2126.978} C_VEL
LIN {X 0,Y 577.944,Z 857.28,A -85,B 0,C 180,E1 2132.965,E2 2132.965} C_VEL
LIN {X 0,Y 578.055,Z 857.28,A -85,B 0,C 180,E1 2138.477,E2 2138.477} C_VEL
LIN {X 0,Y 578.218,Z 857.28,A -85,B 0,C 180,E1 2143.247,E2 2143.247} C_VEL
LIN {X 0,Y 578.181,Z 857.28,A -85,B 0,C 180,E1 2149.423,E2 2149.423} C_VEL
LIN {X 0,Y 578.441,Z 857.28,A -85,B 0,C 180,E1 2154.079,E2 2154.079} C_VEL
LIN {X 0,Y 578.193,Z 857.28,A -85,B 0,C 180,E1 2159.981,E2 2159.981} C_VEL
LIN {X 0,Y 578.243,Z 857.28,A -85,B 0,C 180,E1 2164.484,E2 2164.484} C_VEL
LIN {X 0,Y 578.227,Z 857.28,A -85,B 0,C 180,E1 2169.016,E2 2169.016} C_VEL
LIN {X 0,Y 578.088,Z 857.28,A -85,B 0,C 180,E1 2174.285,E2 2174.285} C_VEL
LIN {X 0,Y 578.075,Z 857.28,A -85,B 0,C 180,E1 2179.877,E2 2179.877} C_VEL
LIN {X 0,Y 577.971,Z 857.28,A -85,B 0,C 180,E1 2184.748,E2 2184.748} C_VEL
LIN {X 0,Y 577.828,Z 857.28,A -85,B 0,C 180,E1 2190.151,E2 2190.151} C_VEL
LIN {X 0,Y 577.856,Z 857.28,A -85,B 0,C 180,E1 2195.159,E2 2195.159} C_VEL
LIN {X 0,Y 577.827,Z 857.28,A -85,B 0,C 180,E1 2200.878,E2 2200.878} C_VEL
LIN {X 0,Y 577.981,Z 857.28,A -85,B 0,C 180,E1 2207.124,E2 2207.124} C_VEL
LIN {X 0,Y 577.962,Z 857.28,A -85,B 0,C 180,E1 2212.948,E2 2212.948} C_VEL
LIN {X 0,Y 578.318,Z 857.965,A -85,B 0,C 180,E1 2218.277,E2 2218.277} C_VEL
LIN {X 0,Y 579.397,Z 882.384,A -85,B 0,C 180,E1 2219.439,E2 2219.439} C_VEL
LIN {X 0,Y 579.105,Z 906.576,A -85,B 0,C 180,E1 2221.14,E2 2221.14} C_VEL
LIN {X 0,Y 578.845,Z 928.007,A -85,B 0,C 180,E1 2223.371,E2 2223.371} C_VEL
LIN {X 0,Y 578.691,Z 943.608,A -85,B 0,C 180,E1 2225.772,E2 2225.772} C_VEL
LIN {X 0,Y 578.562,Z 954.853,A -85,B 0,C 180,E1 2228.507,E2 2228.507} C_VEL
LIN {X 0,Y 578.531,Z 959.147,A -85,B 0,C 180,E1 2230.291,E2 2230.291} C_VEL
LIN {X 0,Y 578.425,Z 961.438,A -85,B 0,C 180,E1 2233.265,E2 2233.265} C_VEL
LIN {X 0,Y 578.501,Z 959.531,A -85,B 0,C 180,E1 2235.381,E2 2235.381} C_VEL
LIN {X 0,Y 578.55,Z 953.212,A -85,B 0,C 180,E1 2237.915,E2 2237.915} C_VEL
LIN {X 0,Y 578.717,Z 941.134,A -85,B 0,C 180,E1 2240.588,E2 2240.588} C_VEL
LIN {X 0,Y 578.883,Z 922.906,A -85,B 0,C 180,E1 2243.156,E2 2243.156} C_VEL
LIN {X 0,Y 579.214,Z 901.054,A -85,B 0,C 180,E1 2245.22,E2 2245.22} C_VEL
LIN {X 0,Y 579.507,Z 875.97,A -85,B 0,C 180,E1 2246.817,E2 2246.817} C_VEL
LIN {X 0,Y 578.693,Z 859.653,A -85,B 0,C 180,E1 2247.563,E2 2247.563} C_VEL
LIN {X 0,Y 578.262,Z 857.28,A -85,B 0,C 180,E1 2247.749,E2 2247.749} C_VEL
LIN {X 0,Y 578.229,Z 857.28,A -85,B 0,C 180,E1 2254.505,E2 2254.505} C_VEL
LIN {X 0,Y 578.212,Z 857.28,A -85,B 0,C 180,E1 2259.039,E2 2259.039} C_VEL
LIN {X 0,Y 578.054,Z 857.28,A -85,B 0,C 180,E1 2264.448,E2 2264.448} C_VEL
LIN {X 0,Y 578.023,Z 857.28,A -85,B 0,C 180,E1 2269.908,E2 2269.908} C_VEL
LIN {X 0,Y 577.921,Z 857.28,A -85,B 0,C 180,E1 2274.782,E2 2274.782} C_VEL
LIN {X 0,Y 577.805,Z 857.28,A -85,B 0,C 180,E1 2280.229,E2 2280.229} C_VEL
LIN {X 0,Y 577.861,Z 857.28,A -85,B 0,C 180,E1 2285.199,E2 2285.199} C_VEL
LIN {X 0,Y 577.785,Z 857.28,A -85,B 0,C 180,E1 2290.928,E2 2290.928} C_VEL
LIN {X 0,Y 578.003,Z 857.28,A -85,B 0,C 180,E1 2297.176,E2 2297.176} C_VEL
LIN {X 0,Y 578.055,Z 857.787,A -85,B 0,C 180,E1 2303.263,E2 2303.263} C_VEL
LIN {X 0,Y 579.446,Z 874.329,A -85,B 0,C 180,E1 2304.008,E2 2304.008} C_VEL
LIN {X 0,Y 579.169,Z 900.818,A -85,B 0,C 180,E1 2305.67,E2 2305.67} C_VEL
LIN {X 0,Y 578.85,Z 923.113,A -85,B 0,C 180,E1 2307.778,E2 2307.778} C_VEL
LIN {X 0,Y 578.718,Z 940.613,A -85,B 0,C 180,E1 2310.229,E2 2310.229} C_VEL
LIN {X 0,Y 578.602,Z 952.652,A -85,B 0,C 180,E1 2312.835,E2 2312.835} C_VEL
LIN {X 0,Y 578.521,Z 959.131,A -85,B 0,C 180,E1 2315.277,E2 2315.277} C_VEL
LIN {X 0,Y 578.452,Z 961.113,A -85,B 0,C 180,E1 2316.914,E2 2316.914} C_VEL
LIN {X 0,Y 578.477,Z 961.379,A -85,B 0,C 180,E1 2318.535,E2 2318.535} C_VEL
LIN {X 0,Y 578.547,Z 958.259,A -85,B 0,C 180,E1 2321.071,E2 2321.071} C_VEL
LIN {X 0,Y 578.626,Z 950.328,A -85,B 0,C 180,E1 2323.69,E2 2323.69} C_VEL
LIN {X 0,Y 578.712,Z 936.165,A -85,B 0,C 180,E1 2326.407,E2 2326.407} C_VEL
LIN {X 0,Y 578.927,Z 918.117,A -85,B 0,C 180,E1 2328.679,E2 2328.679} C_VEL
LIN {X 0,Y 579.22,Z 894.36,A -85,B 0,C 180,E1 2330.716,E2 2330.716} C_VEL
LIN {X 0,Y 579.605,Z 867.126,A -85,B 0,C 180,E1 2332.235,E2 2332.235} C_VEL
LIN {X 0,Y 578.498,Z 857.28,A -85,B 0,C 180,E1 2332.692,E2 2332.692} C_VEL
LIN {X 0,Y 578.421,Z 857.28,A -85,B 0,C 180,E1 2338.52,E2 2338.52} C_VEL
LIN {X 0,Y 578.257,Z 857.28,A -85,B 0,C 180,E1 2344.523,E2 2344.523} C_VEL
LIN {X 0,Y 578.112,Z 857.28,A -85,B 0,C 180,E1 2345.814,E2 2345.814} C_VEL
LIN {X 0,Y 574.273,Z 857.28,A -85,B 0,C 180,E1 2347.51,E2 2347.51} C_VEL
LIN {X 0,Y 570.276,Z 857.28,A -85,B 0,C 180,E1 2349.228,E2 2349.228} C_VEL
LIN {X 0,Y 570.256,Z 857.28,A -85,B 0,C 180,E1 2353.839,E2 2353.839} C_VEL
LIN {X 0,Y 570.236,Z 857.28,A -85,B 0,C 180,E1 2358.592,E2 2358.592} C_VEL
LIN {X 0,Y 570.162,Z 857.28,A -85,B 0,C 180,E1 2363.484,E2 2363.484} C_VEL
LIN {X 0,Y 569.998,Z 857.28,A -85,B 0,C 180,E1 2368.769,E2 2368.769} C_VEL
LIN {X 0,Y 569.962,Z 857.28,A -85,B 0,C 180,E1 2374.564,E2 2374.564} C_VEL
LIN {X 0,Y 569.928,Z 857.28,A -85,B 0,C 180,E1 2379.617,E2 2379.617} C_VEL
LIN {X 0,Y 569.986,Z 857.28,A -85,B 0,C 180,E1 2385.827,E2 2385.827} C_VEL
LIN {X 0,Y 569.994,Z 857.28,A -85,B 0,C 180,E1 2390.394,E2 2390.394} C_VEL
LIN {X 0,Y 569.89,Z 857.28,A -85,B 0,C 180,E1 2395.446,E2 2395.446} C_VEL
LIN {X 0,Y 569.991,Z 857.28,A -85,B 0,C 180,E1 2401.228,E2 2401.228} C_VEL
LIN {X 0,Y 570.187,Z 857.28,A -85,B 0,C 180,E1 2406.614,E2 2406.614} C_VEL
LIN {X 0,Y 573.842,Z 871.85,A -85,B 0,C 180,E1 2406.969,E2 2406.969} C_VEL
LIN {X 0,Y 573.755,Z 938.276,A -85,B 0,C 180,E1 2407.954,E2 2407.954} C_VEL
LIN {X 0,Y 573.17,Z 972.424,A -85,B 0,C 180,E1 2409.058,E2 2409.058} C_VEL
LIN {X 0,Y 572.565,Z 1004.113,A -85,B 0,C 180,E1 2410.699,E2 2410.699} C_VEL
LIN {X 0,Y 571.86,Z 1033.396,A -85,B 0,C 180,E1 2412.883,E2 2412.883} C_VEL
LIN {X 0,Y 571.33,Z 1058.552,A -85,B 0,C 180,E1 2415.477,E2 2415.477} C_VEL
LIN {X 0,Y 570.976,Z 1079.207,A -85,B 0,C 180,E1 2418.394,E2 2418.394} C_VEL
LIN {X 0,Y 570.733,Z 1095.118,A -85,B 0,C 180,E1 2421.611,E2 2421.611} C_VEL
LIN {X 0,Y 570.66,Z 1105.302,A -85,B 0,C 180,E1 2424.797,E2 2424.797} C_VEL
LIN {X 0,Y 570.514,Z 1109.401,A -85,B 0,C 180,E1 2426.958,E2 2426.958} C_VEL
LIN {X 0,Y 570.553,Z 1111.5,A -85,B 0,C 180,E1 2430.001,E2 2430.001} C_VEL
LIN {X 0,Y 570.545,Z 1109.398,A -85,B 0,C 180,E1 2433.043,E2 2433.043} C_VEL
LIN {X 0,Y 570.589,Z 1101.848,A -85,B 0,C 180,E1 2436.476,E2 2436.476} C_VEL
LIN {X 0,Y 570.745,Z 1090.123,A -85,B 0,C 180,E1 2439.544,E2 2439.544} C_VEL
LIN {X 0,Y 570.99,Z 1072.664,A -85,B 0,C 180,E1 2442.637,E2 2442.637} C_VEL
LIN {X 0,Y 571.52,Z 1049.484,A -85,B 0,C 180,E1 2445.56,E2 2445.56} C_VEL
LIN {X 0,Y 572.134,Z 1021.472,A -85,B 0,C 180,E1 2448.097,E2 2448.097} C_VEL
LIN {X 0,Y 572.849,Z 990.275,A -85,B 0,C 180,E1 2450.097,E2 2450.097} C_VEL
LIN {X 0,Y 573.515,Z 957.927,A -85,B 0,C 180,E1 2451.488,E2 2451.488} C_VEL
LIN {X 0,Y 573.851,Z 925.892,A -85,B 0,C 180,E1 2452.294,E2 2452.294} C_VEL
LIN {X 0,Y 573.179,Z 867.442,A -85,B 0,C 180,E1 2453.118,E2 2453.118} C_VEL
LIN {X 0,Y 570.079,Z 857.28,A -85,B 0,C 180,E1 2453.42,E2 2453.42} C_VEL
LIN {X 0,Y 569.997,Z 857.28,A -85,B 0,C 180,E1 2458.773,E2 2458.773} C_VEL
LIN {X 0,Y 569.954,Z 857.28,A -85,B 0,C 180,E1 2464.564,E2 2464.564} C_VEL
LIN {X 0,Y 569.951,Z 857.28,A -85,B 0,C 180,E1 2469.611,E2 2469.611} C_VEL
LIN {X 0,Y 569.966,Z 857.28,A -85,B 0,C 180,E1 2475.828,E2 2475.828} C_VEL
LIN {X 0,Y 569.995,Z 857.28,A -85,B 0,C 180,E1 2480.389,E2 2480.389} C_VEL
LIN {X 0,Y 569.903,Z 857.28,A -85,B 0,C 180,E1 2486.082,E2 2486.082} C_VEL
LIN {X 0,Y 569.96,Z 857.28,A -85,B 0,C 180,E1 2491.426,E2 2491.426} C_VEL
LIN {X 0,Y 570.108,Z 857.28,A -85,B 0,C 180,E1 2496.514,E2 2496.514} C_VEL
LIN {X 0,Y 570.257,Z 857.28,A -85,B 0,C 180,E1 2501.409,E2 2501.409} C_VEL
LIN {X 0,Y 569.857,Z 857.28,A -85,B 0,C 180,E1 2506.151,E2 2506.151} C_VEL
LIN {X 0,Y 570.168,Z 857.28,A -85,B 0,C 180,E1 2510.816,E2 2510.816} C_VEL
LIN {X 0,Y 570.266,Z 857.28,A -85,B 0,C 180,E1 2515.414,E2 2515.414} C_VEL
LIN {X 0,Y 570.306,Z 857.28,A -85,B 0,C 180,E1 2519.981,E2 2519.981} C_VEL
LIN {X 0,Y 570.34,Z 857.28,A -85,B 0,C 180,E1 2524.546,E2 2524.546} C_VEL
LIN {X 0,Y 570.294,Z 857.28,A -85,B 0,C 180,E1 2529.142,E2 2529.142} C_VEL
LIN {X 0,Y 570.273,Z 857.28,A -85,B 0,C 180,E1 2533.798,E2 2533.798} C_VEL
LIN {X 0,Y 570.246,Z 857.28,A -85,B 0,C 180,E1 2538.55,E2 2538.55} C_VEL
LIN {X 0,Y 570.128,Z 857.28,A -85,B 0,C 180,E1 2543.443,E2 2543.443} C_VEL
LIN {X 0,Y 569.99,Z 857.28,A -85,B 0,C 180,E1 2548.766,E2 2548.766} C_VEL
LIN {X 0,Y 569.973,Z 857.28,A -85,B 0,C 180,E1 2554.564,E2 2554.564} C_VEL
LIN {X 0,Y 569.923,Z 857.28,A -85,B 0,C 180,E1 2559.607,E2 2559.607} C_VEL
LIN {X 0,Y 569.997,Z 857.28,A -85,B 0,C 180,E1 2565.77,E2 2565.77} C_VEL
LIN {X 0,Y 569.966,Z 857.28,A -85,B 0,C 180,E1 2570.39,E2 2570.39} C_VEL
LIN {X 0,Y 570.012,Z 857.28,A -85,B 0,C 180,E1 2576.095,E2 2576.095} C_VEL
LIN {X 0,Y 570.392,Z 858.089,A -85,B 0,C 180,E1 2578.072,E2 2578.072} C_VEL
LIN {X 0,Y 571.751,Z 876.685,A -85,B 0,C 180,E1 2578.938,E2 2578.938} C_VEL
LIN {X 0,Y 571.4,Z 901.31,A -85,B 0,C 180,E1 2580.54,E2 2580.54} C_VEL
LIN {X 0,Y 571.076,Z 922.595,A -85,B 0,C 180,E1 2582.576,E2 2582.576} C_VEL
LIN {X 0,Y 570.826,Z 940.665,A -85,B 0,C 180,E1 2585.133,E2 2585.133} C_VEL
LIN {X 0,Y 570.673,Z 952.686,A -85,B 0,C 180,E1 2587.776,E2 2587.776} C_VEL
LIN {X 0,Y 570.592,Z 959.951,A -85,B 0,C 180,E1 2590.764,E2 2590.764} C_VEL
LIN {X 0,Y 570.5,Z 961.492,A -85,B 0,C 180,E1 2593.026,E2 2593.026} C_VEL
LIN {X 0,Y 570.578,Z 959.908,A -85,B 0,C 180,E1 2595.173,E2 2595.173} C_VEL
LIN {X 0,Y 570.674,Z 954.008,A -85,B 0,C 180,E1 2597.745,E2 2597.745} C_VEL
LIN {X 0,Y 570.843,Z 942.472,A -85,B 0,C 180,E1 2600.457,E2 2600.457} C_VEL
LIN {X 0,Y 571.058,Z 925.363,A -85,B 0,C 180,E1 2603.001,E2 2603.001} C_VEL
LIN {X 0,Y 571.423,Z 902.804,A -85,B 0,C 180,E1 2605.25,E2 2605.25} C_VEL
LIN {X 0,Y 571.796,Z 876.818,A -85,B 0,C 180,E1 2606.964,E2 2606.964} C_VEL
LIN {X 0,Y 570.952,Z 860.781,A -85,B 0,C 180,E1 2607.72,E2 2607.72} C_VEL
LIN {X 0,Y 570.312,Z 857.28,A -85,B 0,C 180,E1 2607.907,E2 2607.907} C_VEL
LIN {X 0,Y 570.334,Z 857.28,A -85,B 0,C 180,E1 2614.567,E2 2614.567} C_VEL
LIN {X 0,Y 570.283,Z 857.28,A -85,B 0,C 180,E1 2619.166,E2 2619.166} C_VEL
LIN {X 0,Y 570.278,Z 857.28,A -85,B 0,C 180,E1 2623.824,E2 2623.824} C_VEL
LIN {X 0,Y 570.204,Z 857.28,A -85,B 0,C 180,E1 2628.58,E2 2628.58} C_VEL
LIN {X 0,Y 570.076,Z 857.28,A -85,B 0,C 180,E1 2633.477,E2 2633.477} C_VEL
LIN {X 0,Y 569.947,Z 857.28,A -85,B 0,C 180,E1 2638.844,E2 2638.844} C_VEL
LIN {X 0,Y 569.97,Z 857.28,A -85,B 0,C 180,E1 2644.635,E2 2644.635} C_VEL
LIN {X 0,Y 569.872,Z 857.28,A -85,B 0,C 180,E1 2649.662,E2 2649.662} C_VEL
LIN {X 0,Y 570,Z 857.28,A -85,B 0,C 180,E1 2655.823,E2 2655.823} C_VEL
LIN {X 0,Y 569.915,Z 857.28,A -85,B 0,C 180,E1 2660.433,E2 2660.433} C_VEL
LIN {X 0,Y 570.109,Z 857.645,A -85,B 0,C 180,E1 2663.048,E2 2663.048} C_VEL
LIN {X 0,Y 571.75,Z 874.508,A -85,B 0,C 180,E1 2663.826,E2 2663.826} C_VEL
LIN {X 0,Y 571.428,Z 900.322,A -85,B 0,C 180,E1 2665.462,E2 2665.462} C_VEL
LIN {X 0,Y 571.061,Z 922.809,A -85,B 0,C 180,E1 2667.603,E2 2667.603} C_VEL
LIN {X 0,Y 570.846,Z 940.631,A -85,B 0,C 180,E1 2670.124,E2 2670.124} C_VEL
LIN {X 0,Y 570.718,Z 952.877,A -85,B 0,C 180,E1 2672.828,E2 2672.828} C_VEL
LIN {X 0,Y 570.632,Z 958.493,A -85,B 0,C 180,E1 2674.912,E2 2674.912} C_VEL
LIN {X 0,Y 570.547,Z 960.89,A -85,B 0,C 180,E1 2676.575,E2 2676.575} C_VEL
LIN {X 0,Y 570.544,Z 961.443,A -85,B 0,C 180,E1 2678.249,E2 2678.249} C_VEL
LIN {X 0,Y 570.654,Z 958.81,A -85,B 0,C 180,E1 2680.839,E2 2680.839} C_VEL
LIN {X 0,Y 570.755,Z 949.99,A -85,B 0,C 180,E1 2683.854,E2 2683.854} C_VEL
LIN {X 0,Y 570.872,Z 935.618,A -85,B 0,C 180,E1 2686.607,E2 2686.607} C_VEL
LIN {X 0,Y 571.109,Z 917.002,A -85,B 0,C 180,E1 2688.946,E2 2688.946} C_VEL
LIN {X 0,Y 571.487,Z 893.203,A -85,B 0,C 180,E1 2690.973,E2 2690.973} C_VEL
LIN {X 0,Y 571.939,Z 866.359,A -85,B 0,C 180,E1 2692.464,E2 2692.464} C_VEL
LIN {X 0,Y 570.564,Z 857.28,A -85,B 0,C 180,E1 2692.877,E2 2692.877} C_VEL
LIN {X 0,Y 570.522,Z 857.28,A -85,B 0,C 180,E1 2698.499,E2 2698.499} C_VEL
LIN {X 0,Y 570.354,Z 857.28,A -85,B 0,C 180,E1 2704.585,E2 2704.585} C_VEL
LIN {X 0,Y 570.276,Z 857.28,A -85,B 0,C 180,E1 2709.228,E2 2709.228} C_VEL
LIN {X 0,Y 566.24,Z 857.28,A -85,B 0,C 180,E1 2710.941,E2 2710.941} C_VEL
LIN {X 0,Y 562.292,Z 857.28,A -85,B 0,C 180,E1 2712.678,E2 2712.678} C_VEL
LIN {X 0,Y 562.287,Z 857.28,A -85,B 0,C 180,E1 2718.864,E2 2718.864} C_VEL
LIN {X 0,Y 562.223,Z 857.28,A -85,B 0,C 180,E1 2723.836,E2 2723.836} C_VEL
LIN {X 0,Y 562.063,Z 857.28,A -85,B 0,C 180,E1 2729.013,E2 2729.013} C_VEL
LIN {X 0,Y 562.072,Z 857.28,A -85,B 0,C 180,E1 2734.457,E2 2734.457} C_VEL
LIN {X 0,Y 561.93,Z 857.28,A -85,B 0,C 180,E1 2740.295,E2 2740.295} C_VEL
LIN {X 0,Y 562.074,Z 857.28,A -85,B 0,C 180,E1 2745.544,E2 2745.544} C_VEL
LIN {X 0,Y 562.056,Z 857.28,A -85,B 0,C 180,E1 2751.715,E2 2751.715} C_VEL
LIN {X 0,Y 561.988,Z 857.28,A -85,B 0,C 180,E1 2757.397,E2 2757.397} C_VEL
LIN {X 0,Y 562.128,Z 857.28,A -85,B 0,C 180,E1 2762.75,E2 2762.75} C_VEL
LIN {X 0,Y 562.296,Z 857.424,A -85,B 0,C 180,E1 2766.271,E2 2766.271} C_VEL
LIN {X 0,Y 566.49,Z 870.75,A -85,B 0,C 180,E1 2766.637,E2 2766.637} C_VEL
LIN {X 0,Y 566.402,Z 939.849,A -85,B 0,C 180,E1 2767.693,E2 2767.693} C_VEL
LIN {X 0,Y 565.727,Z 973.653,A -85,B 0,C 180,E1 2768.821,E2 2768.821} C_VEL
LIN {X 0,Y 564.985,Z 1005.646,A -85,B 0,C 180,E1 2770.531,E2 2770.531} C_VEL
LIN {X 0,Y 564.15,Z 1035.505,A -85,B 0,C 180,E1 2772.83,E2 2772.83} C_VEL
LIN {X 0,Y 563.515,Z 1061.446,A -85,B 0,C 180,E1 2775.63,E2 2775.63} C_VEL
LIN {X 0,Y 563.086,Z 1081.889,A -85,B 0,C 180,E1 2778.706,E2 2778.706} C_VEL
LIN {X 0,Y 562.872,Z 1096.652,A -85,B 0,C 180,E1 2781.882,E2 2781.882} C_VEL
LIN {X 0,Y 562.749,Z 1106.728,A -85,B 0,C 180,E1 2785.371,E2 2785.371} C_VEL
LIN {X 0,Y 562.674,Z 1110.933,A -85,B 0,C 180,E1 2788.459,E2 2788.459} C_VEL
LIN {X 0,Y 562.682,Z 1110.932,A -85,B 0,C 180,E1 2791.542,E2 2791.542} C_VEL
LIN {X 0,Y 562.724,Z 1106.725,A -85,B 0,C 180,E1 2794.63,E2 2794.63} C_VEL
LIN {X 0,Y 562.865,Z 1096.649,A -85,B 0,C 180,E1 2798.119,E2 2798.119} C_VEL
LIN {X 0,Y 563.1,Z 1080.34,A -85,B 0,C 180,E1 2801.573,E2 2801.573} C_VEL
LIN {X 0,Y 563.554,Z 1059.732,A -85,B 0,C 180,E1 2804.582,E2 2804.582} C_VEL
LIN {X 0,Y 564.191,Z 1033.857,A -85,B 0,C 180,E1 2807.316,E2 2807.316} C_VEL
LIN {X 0,Y 565.012,Z 1004.092,A -85,B 0,C 180,E1 2809.571,E2 2809.571} C_VEL
LIN {X 0,Y 565.718,Z 971.551,A -85,B 0,C 180,E1 2811.269,E2 2811.269} C_VEL
LIN {X 0,Y 566.347,Z 936.244,A -85,B 0,C 180,E1 2812.397,E2 2812.397} C_VEL
LIN {X 0,Y 565.858,Z 868.999,A -85,B 0,C 180,E1 2813.414,E2 2813.414} C_VEL
LIN {X 0,Y 562.138,Z 857.28,A -85,B 0,C 180,E1 2813.83,E2 2813.83} C_VEL
LIN {X 0,Y 562.083,Z 857.28,A -85,B 0,C 180,E1 2819.004,E2 2819.004} C_VEL
LIN {X 0,Y 562.062,Z 857.28,A -85,B 0,C 180,E1 2824.451,E2 2824.451} C_VEL
LIN {X 0,Y 561.946,Z 857.28,A -85,B 0,C 180,E1 2830.29,E2 2830.29} C_VEL
LIN {X 0,Y 562.034,Z 857.28,A -85,B 0,C 180,E1 2835.536,E2 2835.536} C_VEL
LIN {X 0,Y 562.052,Z 857.28,A -85,B 0,C 180,E1 2841.709,E2 2841.709} C_VEL
LIN {X 0,Y 561.98,Z 857.28,A -85,B 0,C 180,E1 2847.388,E2 2847.388} C_VEL
LIN {X 0,Y 562.09,Z 857.28,A -85,B 0,C 180,E1 2852.737,E2 2852.737} C_VEL
LIN {X 0,Y 562.173,Z 857.28,A -85,B 0,C 180,E1 2857.837,E2 2857.837} C_VEL
LIN {X 0,Y 562.376,Z 857.28,A -85,B 0,C 180,E1 2862.76,E2 2862.76} C_VEL
LIN {X 0,Y 562.337,Z 857.28,A -85,B 0,C 180,E1 2869.121,E2 2869.121} C_VEL
LIN {X 0,Y 562.397,Z 857.28,A -85,B 0,C 180,E1 2874.95,E2 2874.95} C_VEL
LIN {X 0,Y 562.406,Z 857.28,A -85,B 0,C 180,E1 2879.98,E2 2879.98} C_VEL
LIN {X 0,Y 562.378,Z 857.28,A -85,B 0,C 180,E1 2885.028,E2 2885.028} C_VEL
LIN {X 0,Y 562.26,Z 857.28,A -85,B 0,C 180,E1 2890.84,E2 2890.84} C_VEL
LIN {X 0,Y 562.181,Z 857.28,A -85,B 0,C 180,E1 2895.596,E2 2895.596} C_VEL
LIN {X 0,Y 562.218,Z 857.28,A -85,B 0,C 180,E1 2900.463,E2 2900.463} C_VEL
LIN {X 0,Y 562.166,Z 857.28,A -85,B 0,C 180,E1 2905.493,E2 2905.493} C_VEL
LIN {X 0,Y 562.042,Z 857.28,A -85,B 0,C 180,E1 2910.749,E2 2910.749} C_VEL
LIN {X 0,Y 561.984,Z 857.28,A -85,B 0,C 180,E1 2916.307,E2 2916.307} C_VEL
LIN {X 0,Y 561.931,Z 857.28,A -85,B 0,C 180,E1 2922.297,E2 2922.297} C_VEL
LIN {X 0,Y 562.048,Z 857.28,A -85,B 0,C 180,E1 2927.664,E2 2927.664} C_VEL
LIN {X 0,Y 562.123,Z 857.28,A -85,B 0,C 180,E1 2933.838,E2 2933.838} C_VEL
LIN {X 0,Y 562.391,Z 857.879,A -85,B 0,C 180,E1 2937.848,E2 2937.848} C_VEL
LIN {X 0,Y 564.094,Z 875.013,A -85,B 0,C 180,E1 2938.657,E2 2938.657} C_VEL
LIN {X 0,Y 563.659,Z 900.851,A -85,B 0,C 180,E1 2940.33,E2 2940.33} C_VEL
LIN {X 0,Y 563.247,Z 922.496,A -85,B 0,C 180,E1 2942.418,E2 2942.418} C_VEL
LIN {X 0,Y 562.949,Z 940.051,A -85,B 0,C 180,E1 2944.913,E2 2944.913} C_VEL
LIN {X 0,Y 562.794,Z 951.835,A -85,B 0,C 180,E1 2947.457,E2 2947.457} C_VEL
LIN {X 0,Y 562.712,Z 959.148,A -85,B 0,C 180,E1 2950.218,E2 2950.218} C_VEL
LIN {X 0,Y 562.621,Z 961.469,A -85,B 0,C 180,E1 2952.781,E2 2952.781} C_VEL
LIN {X 0,Y 562.7,Z 959.538,A -85,B 0,C 180,E1 2955.444,E2 2955.444} C_VEL
LIN {X 0,Y 562.765,Z 953.093,A -85,B 0,C 180,E1 2958.089,E2 2958.089} C_VEL
LIN {X 0,Y 562.977,Z 940.545,A -85,B 0,C 180,E1 2960.908,E2 2960.908} C_VEL
LIN {X 0,Y 563.215,Z 922.931,A -85,B 0,C 180,E1 2963.44,E2 2963.44} C_VEL
LIN {X 0,Y 563.669,Z 900.975,A -85,B 0,C 180,E1 2965.57,E2 2965.57} C_VEL
LIN {X 0,Y 564.147,Z 875.792,A -85,B 0,C 180,E1 2967.211,E2 2967.211} C_VEL
LIN {X 0,Y 562.83,Z 859.845,A -85,B 0,C 180,E1 2967.976,E2 2967.976} C_VEL
LIN {X 0,Y 562.358,Z 857.28,A -85,B 0,C 180,E1 2968.167,E2 2968.167} C_VEL
LIN {X 0,Y 562.421,Z 857.28,A -85,B 0,C 180,E1 2974.632,E2 2974.632} C_VEL
LIN {X 0,Y 562.383,Z 857.28,A -85,B 0,C 180,E1 2979.295,E2 2979.295} C_VEL
LIN {X 0,Y 562.282,Z 857.28,A -85,B 0,C 180,E1 2984.392,E2 2984.392} C_VEL
LIN {X 0,Y 562.196,Z 857.28,A -85,B 0,C 180,E1 2989.635,E2 2989.635} C_VEL
LIN {X 0,Y 562.098,Z 857.28,A -85,B 0,C 180,E1 2995.529,E2 2995.529} C_VEL
LIN {X 0,Y 561.993,Z 857.28,A -85,B 0,C 180,E1 3000.789,E2 3000.789} C_VEL
LIN {X 0,Y 561.984,Z 857.28,A -85,B 0,C 180,E1 3006.349,E2 3006.349} C_VEL
LIN {X 0,Y 561.896,Z 857.28,A -85,B 0,C 180,E1 3012.348,E2 3012.348} C_VEL
LIN {X 0,Y 562.057,Z 857.28,A -85,B 0,C 180,E1 3017.715,E2 3017.715} C_VEL
LIN {X 0,Y 562.174,Z 857.28,A -85,B 0,C 180,E1 3022.813,E2 3022.813} C_VEL
LIN {X 0,Y 564.064,Z 874.627,A -85,B 0,C 180,E1 3023.635,E2 3023.635} C_VEL
LIN {X 0,Y 563.663,Z 901.016,A -85,B 0,C 180,E1 3025.342,E2 3025.342} C_VEL
LIN {X 0,Y 563.241,Z 923.309,A -85,B 0,C 180,E1 3027.517,E2 3027.517} C_VEL
LIN {X 0,Y 562.973,Z 940.662,A -85,B 0,C 180,E1 3030.018,E2 3030.018} C_VEL
LIN {X 0,Y 562.822,Z 953.09,A -85,B 0,C 180,E1 3032.82,E2 3032.82} C_VEL
LIN {X 0,Y 562.688,Z 959.414,A -85,B 0,C 180,E1 3035.384,E2 3035.384} C_VEL
LIN {X 0,Y 562.614,Z 961.495,A -85,B 0,C 180,E1 3037.898,E2 3037.898} C_VEL
LIN {X 0,Y 562.713,Z 959.692,A -85,B 0,C 180,E1 3040.344,E2 3040.344} C_VEL
LIN {X 0,Y 562.794,Z 952.662,A -85,B 0,C 180,E1 3043.218,E2 3043.218} C_VEL
LIN {X 0,Y 562.958,Z 939.949,A -85,B 0,C 180,E1 3046.019,E2 3046.019} C_VEL
LIN {X 0,Y 563.294,Z 921.265,A -85,B 0,C 180,E1 3048.632,E2 3048.632} C_VEL
LIN {X 0,Y 563.668,Z 898.703,A -85,B 0,C 180,E1 3050.749,E2 3050.749} C_VEL
LIN {X 0,Y 564.212,Z 871.961,A -85,B 0,C 180,E1 3052.407,E2 3052.407} C_VEL
LIN {X 0,Y 562.666,Z 857.28,A -85,B 0,C 180,E1 3053.152,E2 3053.152} C_VEL
LIN {X 0,Y 562.611,Z 857.28,A -85,B 0,C 180,E1 3058.478,E2 3058.478} C_VEL
LIN {X 0,Y 562.438,Z 857.28,A -85,B 0,C 180,E1 3064.65,E2 3064.65} C_VEL
LIN {X 0,Y 562.376,Z 857.28,A -85,B 0,C 180,E1 3069.312,E2 3069.312} C_VEL
LIN {X 0,Y 562.292,Z 857.28,A -85,B 0,C 180,E1 3072.678,E2 3072.678} C_VEL
LIN {X 0,Y 558.208,Z 857.28,A -85,B 0,C 180,E1 3074.416,E2 3074.416} C_VEL
LIN {X 0,Y 554.252,Z 857.28,A -85,B 0,C 180,E1 3076.178,E2 3076.178} C_VEL
LIN {X 0,Y 554.286,Z 857.28,A -85,B 0,C 180,E1 3081.763,E2 3081.763} C_VEL
LIN {X 0,Y 554.187,Z 857.28,A -85,B 0,C 180,E1 3087.684,E2 3087.684} C_VEL
LIN {X 0,Y 554.195,Z 857.28,A -85,B 0,C 180,E1 3093.129,E2 3093.129} C_VEL
LIN {X 0,Y 554.022,Z 857.28,A -85,B 0,C 180,E1 3098.95,E2 3098.95} C_VEL
LIN {X 0,Y 554.168,Z 857.28,A -85,B 0,C 180,E1 3105.268,E2 3105.268} C_VEL
LIN {X 0,Y 554.138,Z 857.28,A -85,B 0,C 180,E1 3111.066,E2 3111.066} C_VEL
LIN {X 0,Y 554.071,Z 857.28,A -85,B 0,C 180,E1 3116.871,E2 3116.871} C_VEL
LIN {X 0,Y 554.218,Z 857.28,A -85,B 0,C 180,E1 3122.328,E2 3122.328} C_VEL
LIN {X 0,Y 554.377,Z 857.28,A -85,B 0,C 180,E1 3125.893,E2 3125.893} C_VEL
LIN {X 0,Y 559.288,Z 873.264,A -85,B 0,C 180,E1 3126.353,E2 3126.353} C_VEL
LIN {X 0,Y 559.101,Z 939.481,A -85,B 0,C 180,E1 3127.376,E2 3127.376} C_VEL
LIN {X 0,Y 558.383,Z 972.429,A -85,B 0,C 180,E1 3128.476,E2 3128.476} C_VEL
LIN {X 0,Y 557.459,Z 1005.37,A -85,B 0,C 180,E1 3130.239,E2 3130.239} C_VEL
LIN {X 0,Y 556.552,Z 1034.07,A -85,B 0,C 180,E1 3132.457,E2 3132.457} C_VEL
LIN {X 0,Y 555.813,Z 1059.716,A -85,B 0,C 180,E1 3135.209,E2 3135.209} C_VEL
LIN {X 0,Y 555.256,Z 1081.093,A -85,B 0,C 180,E1 3138.399,E2 3138.399} C_VEL
LIN {X 0,Y 554.992,Z 1096.652,A -85,B 0,C 180,E1 3141.766,E2 3141.766} C_VEL
LIN {X 0,Y 554.848,Z 1106.728,A -85,B 0,C 180,E1 3145.305,E2 3145.305} C_VEL
LIN {X 0,Y 554.77,Z 1110.933,A -85,B 0,C 180,E1 3148.437,E2 3148.437} C_VEL
LIN {X 0,Y 554.778,Z 1110.932,A -85,B 0,C 180,E1 3151.564,E2 3151.564} C_VEL
LIN {X 0,Y 554.825,Z 1106.725,A -85,B 0,C 180,E1 3154.696,E2 3154.696} C_VEL
LIN {X 0,Y 554.99,Z 1096.649,A -85,B 0,C 180,E1 3158.235,E2 3158.235} C_VEL
LIN {X 0,Y 555.251,Z 1081.087,A -85,B 0,C 180,E1 3161.602,E2 3161.602} C_VEL
LIN {X 0,Y 555.794,Z 1059.732,A -85,B 0,C 180,E1 3164.79,E2 3164.79} C_VEL
LIN {X 0,Y 556.534,Z 1034.075,A -85,B 0,C 180,E1 3167.543,E2 3167.543} C_VEL
LIN {X 0,Y 557.456,Z 1005.248,A -85,B 0,C 180,E1 3169.769,E2 3169.769} C_VEL
LIN {X 0,Y 558.309,Z 972.397,A -85,B 0,C 180,E1 3171.528,E2 3171.528} C_VEL
LIN {X 0,Y 559.041,Z 937.206,A -85,B 0,C 180,E1 3172.685,E2 3172.685} C_VEL
LIN {X 0,Y 558.737,Z 871.197,A -85,B 0,C 180,E1 3173.7,E2 3173.7} C_VEL
LIN {X 0,Y 554.193,Z 857.28,A -85,B 0,C 180,E1 3174.193,E2 3174.193} C_VEL
LIN {X 0,Y 554.161,Z 857.28,A -85,B 0,C 180,E1 3179.459,E2 3179.459} C_VEL
LIN {X 0,Y 554.101,Z 857.28,A -85,B 0,C 180,E1 3185.018,E2 3185.018} C_VEL
LIN {X 0,Y 554.045,Z 857.28,A -85,B 0,C 180,E1 3190.986,E2 3190.986} C_VEL
LIN {X 0,Y 554.149,Z 857.28,A -85,B 0,C 180,E1 3196.912,E2 3196.912} C_VEL
LIN {X 0,Y 554.12,Z 857.28,A -85,B 0,C 180,E1 3203.043,E2 3203.043} C_VEL
LIN {X 0,Y 554.091,Z 857.28,A -85,B 0,C 180,E1 3208.714,E2 3208.714} C_VEL
LIN {X 0,Y 554.295,Z 857.28,A -85,B 0,C 180,E1 3214.345,E2 3214.345} C_VEL
LIN {X 0,Y 554.319,Z 857.28,A -85,B 0,C 180,E1 3219.189,E2 3219.189} C_VEL
LIN {X 0,Y 554.276,Z 857.28,A -85,B 0,C 180,E1 3224.134,E2 3224.134} C_VEL
LIN {X 0,Y 554.374,Z 857.28,A -85,B 0,C 180,E1 3230.552,E2 3230.552} C_VEL
LIN {X 0,Y 554.491,Z 857.28,A -85,B 0,C 180,E1 3235.283,E2 3235.283} C_VEL
LIN {X 0,Y 554.506,Z 857.28,A -85,B 0,C 180,E1 3239.98,E2 3239.98} C_VEL
LIN {X 0,Y 554.532,Z 857.28,A -85,B 0,C 180,E1 3244.676,E2 3244.676} C_VEL
LIN {X 0,Y 554.352,Z 857.28,A -85,B 0,C 180,E1 3250.497,E2 3250.497} C_VEL
LIN {X 0,Y 554.272,Z 857.28,A -85,B 0,C 180,E1 3255.825,E2 3255.825} C_VEL
LIN {X 0,Y 554.275,Z 857.28,A -85,B 0,C 180,E1 3260.769,E2 3260.769} C_VEL
LIN {X 0,Y 554.227,Z 857.28,A -85,B 0,C 180,E1 3265.885,E2 3265.885} C_VEL
LIN {X 0,Y 554.088,Z 857.28,A -85,B 0,C 180,E1 3271.239,E2 3271.239} C_VEL
LIN {X 0,Y 554.003,Z 857.28,A -85,B 0,C 180,E1 3276.916,E2 3276.916} C_VEL
LIN {X 0,Y 554.045,Z 857.28,A -85,B 0,C 180,E1 3283.043,E2 3283.043} C_VEL
LIN {X 0,Y 554.138,Z 857.28,A -85,B 0,C 180,E1 3287.481,E2 3287.481} C_VEL
LIN {X 0,Y 554.13,Z 857.28,A -85,B 0,C 180,E1 3293.049,E2 3293.049} C_VEL
LIN {X 0,Y 554.421,Z 857.503,A -85,B 0,C 180,E1 3297.612,E2 3297.612} C_VEL
LIN {X 0,Y 556.413,Z 874.357,A -85,B 0,C 180,E1 3298.421,E2 3298.421} C_VEL
LIN {X 0,Y 555.922,Z 900.411,A -85,B 0,C 180,E1 3300.116,E2 3300.116} C_VEL
LIN {X 0,Y 555.437,Z 921.857,A -85,B 0,C 180,E1 3302.195,E2 3302.195} C_VEL
LIN {X 0,Y 555.085,Z 939.914,A -85,B 0,C 180,E1 3304.773,E2 3304.773} C_VEL
LIN {X 0,Y 554.901,Z 952.391,A -85,B 0,C 180,E1 3307.542,E2 3307.542} C_VEL
LIN {X 0,Y 554.821,Z 958.691,A -85,B 0,C 180,E1 3309.924,E2 3309.924} C_VEL
LIN {X 0,Y 554.734,Z 961.442,A -85,B 0,C 180,E1 3312.653,E2 3312.653} C_VEL
LIN {X 0,Y 554.828,Z 959.069,A -85,B 0,C 180,E1 3315.782,E2 3315.782} C_VEL
LIN {X 0,Y 554.914,Z 951.491,A -85,B 0,C 180,E1 3318.63,E2 3318.63} C_VEL
LIN {X 0,Y 555.136,Z 938.565,A -85,B 0,C 180,E1 3321.372,E2 3321.372} C_VEL
LIN {X 0,Y 555.462,Z 919.711,A -85,B 0,C 180,E1 3323.958,E2 3323.958} C_VEL
LIN {X 0,Y 555.984,Z 896.57,A -85,B 0,C 180,E1 3326.096,E2 3326.096} C_VEL
LIN {X 0,Y 556.574,Z 869.871,A -85,B 0,C 180,E1 3327.71,E2 3327.71} C_VEL
LIN {X 0,Y 554.445,Z 857.28,A -85,B 0,C 180,E1 3328.337,E2 3328.337} C_VEL
LIN {X 0,Y 554.511,Z 857.28,A -85,B 0,C 180,E1 3334.698,E2 3334.698} C_VEL
LIN {X 0,Y 554.456,Z 857.28,A -85,B 0,C 180,E1 3339.43,E2 3339.43} C_VEL
LIN {X 0,Y 554.42,Z 857.28,A -85,B 0,C 180,E1 3344.228,E2 3344.228} C_VEL
LIN {X 0,Y 554.335,Z 857.28,A -85,B 0,C 180,E1 3349.132,E2 3349.132} C_VEL
LIN {X 0,Y 554.175,Z 857.28,A -85,B 0,C 180,E1 3354.193,E2 3354.193} C_VEL
LIN {X 0,Y 554.092,Z 857.28,A -85,B 0,C 180,E1 3359.462,E2 3359.462} C_VEL
LIN {X 0,Y 554.127,Z 857.28,A -85,B 0,C 180,E1 3365.015,E2 3365.015} C_VEL
LIN {X 0,Y 553.974,Z 857.28,A -85,B 0,C 180,E1 3370.991,E2 3370.991} C_VEL
LIN {X 0,Y 554.151,Z 857.28,A -85,B 0,C 180,E1 3376.967,E2 3376.967} C_VEL
LIN {X 0,Y 554.237,Z 857.28,A -85,B 0,C 180,E1 3382.588,E2 3382.588} C_VEL
LIN {X 0,Y 556.383,Z 875.357,A -85,B 0,C 180,E1 3383.472,E2 3383.472} C_VEL
LIN {X 0,Y 555.914,Z 900.918,A -85,B 0,C 180,E1 3385.155,E2 3385.155} C_VEL
LIN {X 0,Y 555.405,Z 923.44,A -85,B 0,C 180,E1 3387.384,E2 3387.384} C_VEL
LIN {X 0,Y 555.091,Z 941.245,A -85,B 0,C 180,E1 3390.011,E2 3390.011} C_VEL
LIN {X 0,Y 554.937,Z 953.398,A -85,B 0,C 180,E1 3392.841,E2 3392.841} C_VEL
LIN {X 0,Y 554.777,Z 960.179,A -85,B 0,C 180,E1 3395.868,E2 3395.868} C_VEL
LIN {X 0,Y 554.692,Z 961.47,A -85,B 0,C 180,E1 3398.133,E2 3398.133} C_VEL
LIN {X 0,Y 554.839,Z 958.82,A -85,B 0,C 180,E1 3400.915,E2 3400.915} C_VEL
LIN {X 0,Y 554.973,Z 950.707,A -85,B 0,C 180,E1 3403.835,E2 3403.835} C_VEL
LIN {X 0,Y 555.139,Z 937.073,A -85,B 0,C 180,E1 3406.622,E2 3406.622} C_VEL
LIN {X 0,Y 555.453,Z 919.139,A -85,B 0,C 180,E1 3409.025,E2 3409.025} C_VEL
LIN {X 0,Y 555.947,Z 896.318,A -85,B 0,C 180,E1 3411.113,E2 3411.113} C_VEL
LIN {X 0,Y 556.553,Z 870.181,A -85,B 0,C 180,E1 3412.697,E2 3412.697} C_VEL
LIN {X 0,Y 554.765,Z 857.28,A -85,B 0,C 180,E1 3413.362,E2 3413.362} C_VEL
LIN {X 0,Y 554.701,Z 857.28,A -85,B 0,C 180,E1 3418.457,E2 3418.457} C_VEL
LIN {X 0,Y 554.543,Z 857.28,A -85,B 0,C 180,E1 3424.716,E2 3424.716} C_VEL
LIN {X 0,Y 554.346,Z 857.28,A -85,B 0,C 180,E1 3430.5,E2 3430.5} C_VEL
LIN {X 0,Y 554.252,Z 857.28,A -85,B 0,C 180,E1 3436.178,E2 3436.178} C_VEL
LIN {X 0,Y 551.826,Z 857.28,A -85,B 0,C 180,E1 3437.509,E2 3437.509} C_VEL
LIN {X 0,Y 546.409,Z 857.28,A -85,B 0,C 180,E1 3439.733,E2 3439.733} C_VEL
LIN {X 0,Y 546.336,Z 857.28,A -85,B 0,C 180,E1 3444.574,E2 3444.574} C_VEL
LIN {X 0,Y 546.166,Z 857.28,A -85,B 0,C 180,E1 3449.943,E2 3449.943} C_VEL
LIN {X 0,Y 546.128,Z 857.28,A -85,B 0,C 180,E1 3455.613,E2 3455.613} C_VEL
LIN {X 0,Y 546.136,Z 857.28,A -85,B 0,C 180,E1 3461.715,E2 3461.715} C_VEL
LIN {X 0,Y 546.232,Z 857.28,A -85,B 0,C 180,E1 3466.136,E2 3466.136} C_VEL
LIN {X 0,Y 546.214,Z 857.28,A -85,B 0,C 180,E1 3472.424,E2 3472.424} C_VEL
LIN {X 0,Y 546.183,Z 857.28,A -85,B 0,C 180,E1 3478.218,E2 3478.218} C_VEL
LIN {X 0,Y 546.36,Z 857.28,A -85,B 0,C 180,E1 3483.68,E2 3483.68} C_VEL
LIN {X 0,Y 546.462,Z 857.874,A -85,B 0,C 180,E1 3485.545,E2 3485.545} C_VEL
LIN {X 0,Y 552.093,Z 877.01,A -85,B 0,C 180,E1 3486.078,E2 3486.078} C_VEL
LIN {X 0,Y 551.827,Z 939.48,A -85,B 0,C 180,E1 3487.061,E2 3487.061} C_VEL
LIN {X 0,Y 551.016,Z 972.431,A -85,B 0,C 180,E1 3488.173,E2 3488.173} C_VEL
LIN {X 0,Y 550.033,Z 1003.953,A -85,B 0,C 180,E1 3489.864,E2 3489.864} C_VEL
LIN {X 0,Y 548.957,Z 1032.608,A -85,B 0,C 180,E1 3492.073,E2 3492.073} C_VEL
LIN {X 0,Y 548.061,Z 1058.664,A -85,B 0,C 180,E1 3494.86,E2 3494.86} C_VEL
LIN {X 0,Y 547.434,Z 1080.003,A -85,B 0,C 180,E1 3498.029,E2 3498.029} C_VEL
LIN {X 0,Y 547.11,Z 1095.118,A -85,B 0,C 180,E1 3501.246,E2 3501.246} C_VEL
LIN {X 0,Y 546.945,Z 1105.183,A -85,B 0,C 180,E1 3504.52,E2 3504.52} C_VEL
LIN {X 0,Y 546.839,Z 1109.403,A -85,B 0,C 180,E1 3506.826,E2 3506.826} C_VEL
LIN {X 0,Y 546.885,Z 1111.5,A -85,B 0,C 180,E1 3510.001,E2 3510.001} C_VEL
LIN {X 0,Y 546.861,Z 1109.4,A -85,B 0,C 180,E1 3513.175,E2 3513.175} C_VEL
LIN {X 0,Y 546.94,Z 1101.849,A -85,B 0,C 180,E1 3516.757,E2 3516.757} C_VEL
LIN {X 0,Y 547.162,Z 1088.828,A -85,B 0,C 180,E1 3520.25,E2 3520.25} C_VEL
LIN {X 0,Y 547.68,Z 1070,A -85,B 0,C 180,E1 3523.591,E2 3523.591} C_VEL
LIN {X 0,Y 548.432,Z 1047.585,A -85,B 0,C 180,E1 3526.438,E2 3526.438} C_VEL
LIN {X 0,Y 549.457,Z 1019.896,A -85,B 0,C 180,E1 3529.001,E2 3529.001} C_VEL
LIN {X 0,Y 550.524,Z 988.38,A -85,B 0,C 180,E1 3531.055,E2 3531.055} C_VEL
LIN {X 0,Y 551.48,Z 954.817,A -85,B 0,C 180,E1 3532.499,E2 3532.499} C_VEL
LIN {X 0,Y 552.009,Z 921.749,A -85,B 0,C 180,E1 3533.295,E2 3533.295} C_VEL
LIN {X 0,Y 551.645,Z 873.407,A -85,B 0,C 180,E1 3533.993,E2 3533.993} C_VEL
LIN {X 0,Y 546.285,Z 857.28,A -85,B 0,C 180,E1 3534.566,E2 3534.566} C_VEL
LIN {X 0,Y 546.189,Z 857.28,A -85,B 0,C 180,E1 3539.933,E2 3539.933} C_VEL
LIN {X 0,Y 546.113,Z 857.28,A -85,B 0,C 180,E1 3545.607,E2 3545.607} C_VEL
LIN {X 0,Y 546.135,Z 857.28,A -85,B 0,C 180,E1 3551.711,E2 3551.711} C_VEL
LIN {X 0,Y 546.193,Z 857.28,A -85,B 0,C 180,E1 3556.127,E2 3556.127} C_VEL
LIN {X 0,Y 546.219,Z 857.28,A -85,B 0,C 180,E1 3562.417,E2 3562.417} C_VEL
LIN {X 0,Y 546.171,Z 857.28,A -85,B 0,C 180,E1 3568.208,E2 3568.208} C_VEL
LIN {X 0,Y 546.274,Z 857.28,A -85,B 0,C 180,E1 3573.665,E2 3573.665} C_VEL
LIN {X 0,Y 546.417,Z 857.28,A -85,B 0,C 180,E1 3578.874,E2 3578.874} C_VEL
LIN {X 0,Y 546.392,Z 857.28,A -85,B 0,C 180,E1 3583.899,E2 3583.899} C_VEL
LIN {X 0,Y 546.475,Z 857.28,A -85,B 0,C 180,E1 3590.414,E2 3590.414} C_VEL
LIN {X 0,Y 546.562,Z 857.28,A -85,B 0,C 180,E1 3595.77,E2 3595.77} C_VEL
LIN {X 0,Y 546.605,Z 857.28,A -85,B 0,C 180,E1 3599.98,E2 3599.98} C_VEL
LIN {X 0,Y 546.617,Z 857.28,A -85,B 0,C 180,E1 3604.744,E2 3604.744} C_VEL
LIN {X 0,Y 546.534,Z 857.28,A -85,B 0,C 180,E1 3609.543,E2 3609.543} C_VEL
LIN {X 0,Y 546.491,Z 857.28,A -85,B 0,C 180,E1 3614.412,E2 3614.412} C_VEL
LIN {X 0,Y 546.418,Z 857.28,A -85,B 0,C 180,E1 3619.589,E2 3619.589} C_VEL
LIN {X 0,Y 546.317,Z 857.28,A -85,B 0,C 180,E1 3624.531,E2 3624.531} C_VEL
LIN {X 0,Y 546.164,Z 857.28,A -85,B 0,C 180,E1 3629.896,E2 3629.896} C_VEL
LIN {X 0,Y 546.129,Z 857.28,A -85,B 0,C 180,E1 3635.563,E2 3635.563} C_VEL
LIN {X 0,Y 546.101,Z 857.28,A -85,B 0,C 180,E1 3641.664,E2 3641.664} C_VEL
LIN {X 0,Y 546.198,Z 857.28,A -85,B 0,C 180,E1 3646.131,E2 3646.131} C_VEL
LIN {X 0,Y 546.216,Z 857.28,A -85,B 0,C 180,E1 3652.422,E2 3652.422} C_VEL
LIN {X 0,Y 546.481,Z 857.965,A -85,B 0,C 180,E1 3657.321,E2 3657.321} C_VEL
LIN {X 0,Y 548.819,Z 874.995,A -85,B 0,C 180,E1 3658.211,E2 3658.211} C_VEL
LIN {X 0,Y 548.209,Z 900.206,A -85,B 0,C 180,E1 3659.912,E2 3659.912} C_VEL
LIN {X 0,Y 547.609,Z 922.646,A -85,B 0,C 180,E1 3662.132,E2 3662.132} C_VEL
LIN {X 0,Y 547.234,Z 940.831,A -85,B 0,C 180,E1 3664.824,E2 3664.824} C_VEL
LIN {X 0,Y 547.004,Z 953.226,A -85,B 0,C 180,E1 3667.712,E2 3667.712} C_VEL
LIN {X 0,Y 546.866,Z 959.843,A -85,B 0,C 180,E1 3670.595,E2 3670.595} C_VEL
LIN {X 0,Y 546.797,Z 961.358,A -85,B 0,C 180,E1 3672.266,E2 3672.266} C_VEL
LIN {X 0,Y 546.882,Z 959.535,A -85,B 0,C 180,E1 3675.517,E2 3675.517} C_VEL
LIN {X 0,Y 547.003,Z 952.468,A -85,B 0,C 180,E1 3678.423,E2 3678.423} C_VEL
LIN {X 0,Y 547.258,Z 939.956,A -85,B 0,C 180,E1 3681.247,E2 3681.247} C_VEL
LIN {X 0,Y 547.616,Z 922.227,A -85,B 0,C 180,E1 3683.828,E2 3683.828} C_VEL
LIN {X 0,Y 548.19,Z 899.636,A -85,B 0,C 180,E1 3686.04,E2 3686.04} C_VEL
LIN {X 0,Y 548.895,Z 874.335,A -85,B 0,C 180,E1 3687.727,E2 3687.727} C_VEL
LIN {X 0,Y 546.461,Z 857.28,A -85,B 0,C 180,E1 3688.61,E2 3688.61} C_VEL
LIN {X 0,Y 546.592,Z 857.28,A -85,B 0,C 180,E1 3694.847,E2 3694.847} C_VEL
LIN {X 0,Y 546.536,Z 857.28,A -85,B 0,C 180,E1 3699.567,E2 3699.567} C_VEL
LIN {X 0,Y 546.489,Z 857.28,A -85,B 0,C 180,E1 3704.438,E2 3704.438} C_VEL
LIN {X 0,Y 546.356,Z 857.28,A -85,B 0,C 180,E1 3709.703,E2 3709.703} C_VEL
LIN {X 0,Y 546.256,Z 857.28,A -85,B 0,C 180,E1 3714.567,E2 3714.567} C_VEL
LIN {X 0,Y 546.128,Z 857.28,A -85,B 0,C 180,E1 3719.935,E2 3719.935} C_VEL
LIN {X 0,Y 546.118,Z 857.28,A -85,B 0,C 180,E1 3725.606,E2 3725.606} C_VEL
LIN {X 0,Y 546.059,Z 857.28,A -85,B 0,C 180,E1 3731.717,E2 3731.717} C_VEL
LIN {X 0,Y 546.202,Z 857.28,A -85,B 0,C 180,E1 3736.184,E2 3736.184} C_VEL
LIN {X 0,Y 546.289,Z 857.518,A -85,B 0,C 180,E1 3742.365,E2 3742.365} C_VEL
LIN {X 0,Y 548.695,Z 876.045,A -85,B 0,C 180,E1 3743.298,E2 3743.298} C_VEL
LIN {X 0,Y 548.146,Z 902.022,A -85,B 0,C 180,E1 3745.065,E2 3745.065} C_VEL
LIN {X 0,Y 547.557,Z 924.691,A -85,B 0,C 180,E1 3747.384,E2 3747.384} C_VEL
LIN {X 0,Y 547.231,Z 941.205,A -85,B 0,C 180,E1 3749.89,E2 3749.89} C_VEL
LIN {X 0,Y 547.047,Z 953.119,A -85,B 0,C 180,E1 3752.682,E2 3752.682} C_VEL
LIN {X 0,Y 546.894,Z 959.69,A -85,B 0,C 180,E1 3755.497,E2 3755.497} C_VEL
LIN {X 0,Y 546.781,Z 961.342,A -85,B 0,C 180,E1 3757.223,E2 3757.223} C_VEL
LIN {X 0,Y 546.884,Z 959.9,A -85,B 0,C 180,E1 3760.271,E2 3760.271} C_VEL
LIN {X 0,Y 547.048,Z 952.975,A -85,B 0,C 180,E1 3763.273,E2 3763.273} C_VEL
LIN {X 0,Y 547.233,Z 940.122,A -85,B 0,C 180,E1 3766.221,E2 3766.221} C_VEL
LIN {X 0,Y 547.631,Z 921.874,A -85,B 0,C 180,E1 3768.866,E2 3768.866} C_VEL
LIN {X 0,Y 548.141,Z 899.105,A -85,B 0,C 180,E1 3771.086,E2 3771.086} C_VEL
LIN {X 0,Y 548.878,Z 872.57,A -85,B 0,C 180,E1 3772.793,E2 3772.793} C_VEL
LIN {X 0,Y 546.87,Z 857.28,A -85,B 0,C 180,E1 3773.565,E2 3773.565} C_VEL
LIN {X 0,Y 546.61,Z 857.28,A -85,B 0,C 180,E1 3780.02,E2 3780.02} C_VEL
LIN {X 0,Y 546.63,Z 857.28,A -85,B 0,C 180,E1 3784.785,E2 3784.785} C_VEL
LIN {X 0,Y 546.528,Z 857.28,A -85,B 0,C 180,E1 3789.585,E2 3789.585} C_VEL
LIN {X 0,Y 546.47,Z 857.28,A -85,B 0,C 180,E1 3794.454,E2 3794.454} C_VEL
LIN {X 0,Y 546.409,Z 857.28,A -85,B 0,C 180,E1 3799.733,E2 3799.733} C_VEL
LIN {X 0,Y 542.438,Z 857.28,A -85,B 0,C 180,E1 3801.528,E2 3801.528} C_VEL
LIN {X 0,Y 538.411,Z 857.28,A -85,B 0,C 180,E1 3803.348,E2 3803.348} C_VEL
LIN {X 0,Y 538.249,Z 857.28,A -85,B 0,C 180,E1 3809.307,E2 3809.307} C_VEL
LIN {X 0,Y 538.204,Z 857.28,A -85,B 0,C 180,E1 3815.331,E2 3815.331} C_VEL
LIN {X 0,Y 538.148,Z 857.28,A -85,B 0,C 180,E1 3820.568,E2 3820.568} C_VEL
LIN {X 0,Y 538.253,Z 857.28,A -85,B 0,C 180,E1 3827.005,E2 3827.005} C_VEL
LIN {X 0,Y 538.31,Z 857.28,A -85,B 0,C 180,E1 3831.958,E2 3831.958} C_VEL
LIN {X 0,Y 538.209,Z 857.28,A -85,B 0,C 180,E1 3837.69,E2 3837.69} C_VEL
LIN {X 0,Y 538.434,Z 857.28,A -85,B 0,C 180,E1 3843.262,E2 3843.262} C_VEL
LIN {X 0,Y 538.5,Z 857.28,A -85,B 0,C 180,E1 3845.131,E2 3845.131} C_VEL
LIN {X 0,Y 544.879,Z 877.435,A -85,B 0,C 180,E1 3845.747,E2 3845.747} C_VEL
LIN {X 0,Y 544.545,Z 940.261,A -85,B 0,C 180,E1 3846.758,E2 3846.758} C_VEL
LIN {X 0,Y 543.599,Z 973.64,A -85,B 0,C 180,E1 3847.914,E2 3847.914} C_VEL
LIN {X 0,Y 542.437,Z 1006.223,A -85,B 0,C 180,E1 3849.727,E2 3849.727} C_VEL
LIN {X 0,Y 541.247,Z 1035.502,A -85,B 0,C 180,E1 3852.079,E2 3852.079} C_VEL
LIN {X 0,Y 540.288,Z 1059.837,A -85,B 0,C 180,E1 3854.789,E2 3854.789} C_VEL
LIN {X 0,Y 539.592,Z 1081.095,A -85,B 0,C 180,E1 3858.057,E2 3858.057} C_VEL
LIN {X 0,Y 539.251,Z 1096.651,A -85,B 0,C 180,E1 3861.524,E2 3861.524} C_VEL
LIN {X 0,Y 539.07,Z 1106.727,A -85,B 0,C 180,E1 3865.167,E2 3865.167} C_VEL
LIN {X 0,Y 538.977,Z 1110.933,A -85,B 0,C 180,E1 3868.391,E2 3868.391} C_VEL
LIN {X 0,Y 538.986,Z 1110.932,A -85,B 0,C 180,E1 3871.61,E2 3871.61} C_VEL
LIN {X 0,Y 539.071,Z 1106.724,A -85,B 0,C 180,E1 3874.834,E2 3874.834} C_VEL
LIN {X 0,Y 539.243,Z 1096.648,A -85,B 0,C 180,E1 3878.477,E2 3878.477} C_VEL
LIN {X 0,Y 539.58,Z 1081.089,A -85,B 0,C 180,E1 3881.944,E2 3881.944} C_VEL
LIN {X 0,Y 540.285,Z 1059.845,A -85,B 0,C 180,E1 3885.21,E2 3885.21} C_VEL
LIN {X 0,Y 541.308,Z 1033.676,A -85,B 0,C 180,E1 3888.09,E2 3888.09} C_VEL
LIN {X 0,Y 542.535,Z 1003.906,A -85,B 0,C 180,E1 3890.43,E2 3890.43} C_VEL
LIN {X 0,Y 543.61,Z 971.185,A -85,B 0,C 180,E1 3892.195,E2 3892.195} C_VEL
LIN {X 0,Y 544.501,Z 936.174,A -85,B 0,C 180,E1 3893.349,E2 3893.349} C_VEL
LIN {X 0,Y 544.268,Z 874.803,A -85,B 0,C 180,E1 3894.32,E2 3894.32} C_VEL
LIN {X 0,Y 538.329,Z 857.28,A -85,B 0,C 180,E1 3894.954,E2 3894.954} C_VEL
LIN {X 0,Y 538.271,Z 857.28,A -85,B 0,C 180,E1 3900.419,E2 3900.419} C_VEL
LIN {X 0,Y 538.19,Z 857.28,A -85,B 0,C 180,E1 3906.214,E2 3906.214} C_VEL
LIN {X 0,Y 538.148,Z 857.28,A -85,B 0,C 180,E1 3912.473,E2 3912.473} C_VEL
LIN {X 0,Y 538.213,Z 857.28,A -85,B 0,C 180,E1 3917.528,E2 3917.528} C_VEL
LIN {X 0,Y 538.252,Z 857.28,A -85,B 0,C 180,E1 3923.785,E2 3923.785} C_VEL
LIN {X 0,Y 538.267,Z 857.28,A -85,B 0,C 180,E1 3929.572,E2 3929.572} C_VEL
LIN {X 0,Y 538.393,Z 857.28,A -85,B 0,C 180,E1 3935.039,E2 3935.039} C_VEL
LIN {X 0,Y 538.549,Z 857.28,A -85,B 0,C 180,E1 3940.27,E2 3940.27} C_VEL
LIN {X 0,Y 538.325,Z 857.28,A -85,B 0,C 180,E1 3945.322,E2 3945.322} C_VEL
LIN {X 0,Y 538.555,Z 857.28,A -85,B 0,C 180,E1 3950.272,E2 3950.272} C_VEL
LIN {X 0,Y 538.711,Z 857.28,A -85,B 0,C 180,E1 3955.145,E2 3955.145} C_VEL
LIN {X 0,Y 538.723,Z 857.28,A -85,B 0,C 180,E1 3959.979,E2 3959.979} C_VEL
LIN {X 0,Y 538.703,Z 857.28,A -85,B 0,C 180,E1 3964.814,E2 3964.814} C_VEL
LIN {X 0,Y 538.544,Z 857.28,A -85,B 0,C 180,E1 3970.26,E2 3970.26} C_VEL
LIN {X 0,Y 538.481,Z 857.28,A -85,B 0,C 180,E1 3976.302,E2 3976.302} C_VEL
LIN {X 0,Y 538.385,Z 857.28,A -85,B 0,C 180,E1 3981.866,E2 3981.866} C_VEL
LIN {X 0,Y 538.382,Z 857.28,A -85,B 0,C 180,E1 3986.706,E2 3986.706} C_VEL
LIN {X 0,Y 538.225,Z 857.28,A -85,B 0,C 180,E1 3992.442,E2 3992.442} C_VEL
LIN {X 0,Y 538.176,Z 857.28,A -85,B 0,C 180,E1 3998.193,E2 3998.193} C_VEL
LIN {X 0,Y 538.194,Z 857.28,A -85,B 0,C 180,E1 4004.64,E2 4004.64} C_VEL
LIN {X 0,Y 538.208,Z 857.28,A -85,B 0,C 180,E1 4009.681,E2 4009.681} C_VEL
LIN {X 0,Y 538.338,Z 857.28,A -85,B 0,C 180,E1 4015.77,E2 4015.77} C_VEL
LIN {X 0,Y 538.508,Z 857.779,A -85,B 0,C 180,E1 4016.984,E2 4016.984} C_VEL
LIN {X 0,Y 541.348,Z 874.953,A -85,B 0,C 180,E1 4017.899,E2 4017.899} C_VEL
LIN {X 0,Y 540.685,Z 900.687,A -85,B 0,C 180,E1 4019.644,E2 4019.644} C_VEL
LIN {X 0,Y 539.904,Z 921.817,A -85,B 0,C 180,E1 4021.782,E2 4021.782} C_VEL
LIN {X 0,Y 539.409,Z 939.619,A -85,B 0,C 180,E1 4024.45,E2 4024.45} C_VEL
LIN {X 0,Y 539.134,Z 952.374,A -85,B 0,C 180,E1 4027.378,E2 4027.378} C_VEL
LIN {X 0,Y 539.014,Z 959.451,A -85,B 0,C 180,E1 4030.301,E2 4030.301} C_VEL
LIN {X 0,Y 538.872,Z 961.444,A -85,B 0,C 180,E1 4032.656,E2 4032.656} C_VEL
LIN {X 0,Y 539.039,Z 958.424,A -85,B 0,C 180,E1 4036.212,E2 4036.212} C_VEL
LIN {X 0,Y 539.217,Z 950.324,A -85,B 0,C 180,E1 4039.108,E2 4039.108} C_VEL
LIN {X 0,Y 539.496,Z 935.758,A -85,B 0,C 180,E1 4042.136,E2 4042.136} C_VEL
LIN {X 0,Y 540.115,Z 917.081,A -85,B 0,C 180,E1 4044.67,E2 4044.67} C_VEL
LIN {X 0,Y 540.837,Z 893.911,A -85,B 0,C 180,E1 4046.79,E2 4046.79} C_VEL
LIN {X 0,Y 541.113,Z 869.317,A -85,B 0,C 180,E1 4048.296,E2 4048.296} C_VEL
LIN {X 0,Y 538.475,Z 857.28,A -85,B 0,C 180,E1 4048.992,E2 4048.992} C_VEL
LIN {X 0,Y 538.72,Z 857.28,A -85,B 0,C 180,E1 4054.836,E2 4054.836} C_VEL
LIN {X 0,Y 538.566,Z 857.28,A -85,B 0,C 180,E1 4060.526,E2 4060.526} C_VEL
LIN {X 0,Y 538.46,Z 857.28,A -85,B 0,C 180,E1 4066.33,E2 4066.33} C_VEL
LIN {X 0,Y 538.335,Z 857.28,A -85,B 0,C 180,E1 4071.972,E2 4071.972} C_VEL
LIN {X 0,Y 538.304,Z 857.28,A -85,B 0,C 180,E1 4076.745,E2 4076.745} C_VEL
LIN {X 0,Y 538.201,Z 857.28,A -85,B 0,C 180,E1 4082.516,E2 4082.516} C_VEL
LIN {X 0,Y 538.16,Z 857.28,A -85,B 0,C 180,E1 4088.239,E2 4088.239} C_VEL
LIN {X 0,Y 538.183,Z 857.28,A -85,B 0,C 180,E1 4094.694,E2 4094.694} C_VEL
LIN {X 0,Y 538.197,Z 857.28,A -85,B 0,C 180,E1 4099.729,E2 4099.729} C_VEL
LIN {X 0,Y 538.364,Z 857.28,A -85,B 0,C 180,E1 4102.095,E2 4102.095} C_VEL
LIN {X 0,Y 541.089,Z 877.418,A -85,B 0,C 180,E1 4103.122,E2 4103.122} C_VEL
LIN {X 0,Y 540.48,Z 902.642,A -85,B 0,C 180,E1 4104.88,E2 4104.88} C_VEL
LIN {X 0,Y 539.788,Z 923.276,A -85,B 0,C 180,E1 4107.021,E2 4107.021} C_VEL
LIN {X 0,Y 539.377,Z 940.777,A -85,B 0,C 180,E1 4109.689,E2 4109.689} C_VEL
LIN {X 0,Y 539.154,Z 953.251,A -85,B 0,C 180,E1 4112.647,E2 4112.647} C_VEL
LIN {X 0,Y 539.01,Z 959.185,A -85,B 0,C 180,E1 4115.114,E2 4115.114} C_VEL
LIN {X 0,Y 538.846,Z 961.496,A -85,B 0,C 180,E1 4118.009,E2 4118.009} C_VEL
LIN {X 0,Y 539.07,Z 958.473,A -85,B 0,C 180,E1 4121.186,E2 4121.186} C_VEL
LIN {X 0,Y 539.223,Z 950.219,A -85,B 0,C 180,E1 4124.14,E2 4124.14} C_VEL
LIN {X 0,Y 539.49,Z 936.007,A -85,B 0,C 180,E1 4127.052,E2 4127.052} C_VEL
LIN {X 0,Y 540.05,Z 916.726,A -85,B 0,C 180,E1 4129.672,E2 4129.672} C_VEL
LIN {X 0,Y 540.743,Z 893.415,A -85,B 0,C 180,E1 4131.774,E2 4131.774} C_VEL
LIN {X 0,Y 540.896,Z 867.893,A -85,B 0,C 180,E1 4133.292,E2 4133.292} C_VEL
LIN {X 0,Y 538.933,Z 857.28,A -85,B 0,C 180,E1 4133.875,E2 4133.875} C_VEL
LIN {X 0,Y 538.727,Z 857.28,A -85,B 0,C 180,E1 4140.021,E2 4140.021} C_VEL
LIN {X 0,Y 538.716,Z 857.28,A -85,B 0,C 180,E1 4144.855,E2 4144.855} C_VEL
LIN {X 0,Y 538.532,Z 857.28,A -85,B 0,C 180,E1 4150.26,E2 4150.26} C_VEL
LIN {X 0,Y 538.528,Z 857.28,A -85,B 0,C 180,E1 4154.672,E2 4154.672} C_VEL
LIN {X 0,Y 538.522,Z 857.28,A -85,B 0,C 180,E1 4159.731,E2 4159.731} C_VEL
LIN {X 0,Y 538.411,Z 857.28,A -85,B 0,C 180,E1 4163.348,E2 4163.348} C_VEL
LIN {X 0,Y 534.283,Z 857.28,A -85,B 0,C 180,E1 4165.166,E2 4165.166} C_VEL
LIN {X 0,Y 530.352,Z 857.28,A -85,B 0,C 180,E1 4167.012,E2 4167.012} C_VEL
LIN {X 0,Y 530.322,Z 857.28,A -85,B 0,C 180,E1 4172.86,E2 4172.86} C_VEL
LIN {X 0,Y 530.212,Z 857.28,A -85,B 0,C 180,E1 4178.927,E2 4178.927} C_VEL
LIN {X 0,Y 530.293,Z 857.28,A -85,B 0,C 180,E1 4184.456,E2 4184.456} C_VEL
LIN {X 0,Y 530.31,Z 857.28,A -85,B 0,C 180,E1 4190.435,E2 4190.435} C_VEL
LIN {X 0,Y 530.292,Z 857.28,A -85,B 0,C 180,E1 4195.895,E2 4195.895} C_VEL
LIN {X 0,Y 530.415,Z 857.28,A -85,B 0,C 180,E1 4202.237,E2 4202.237} C_VEL
LIN {X 0,Y 530.567,Z 857.28,A -85,B 0,C 180,E1 4204.747,E2 4204.747} C_VEL
LIN {X 0,Y 537.684,Z 880.479,A -85,B 0,C 180,E1 4205.445,E2 4205.445} C_VEL
LIN {X 0,Y 537.282,Z 940.261,A -85,B 0,C 180,E1 4206.425,E2 4206.425} C_VEL
LIN {X 0,Y 536.251,Z 973.643,A -85,B 0,C 180,E1 4207.595,E2 4207.595} C_VEL
LIN {X 0,Y 535.011,Z 1005.278,A -85,B 0,C 180,E1 4209.367,E2 4209.367} C_VEL
LIN {X 0,Y 533.66,Z 1034.515,A -85,B 0,C 180,E1 4211.72,E2 4211.72} C_VEL
LIN {X 0,Y 532.579,Z 1059.68,A -85,B 0,C 180,E1 4214.543,E2 4214.543} C_VEL
LIN {X 0,Y 531.742,Z 1081.096,A -85,B 0,C 180,E1 4217.879,E2 4217.879} C_VEL
LIN {X 0,Y 531.381,Z 1096.651,A -85,B 0,C 180,E1 4221.397,E2 4221.397} C_VEL
LIN {X 0,Y 531.195,Z 1106.727,A -85,B 0,C 180,E1 4225.095,E2 4225.095} C_VEL
LIN {X 0,Y 531.074,Z 1110.933,A -85,B 0,C 180,E1 4228.367,E2 4228.367} C_VEL
LIN {X 0,Y 531.083,Z 1110.932,A -85,B 0,C 180,E1 4231.634,E2 4231.634} C_VEL
LIN {X 0,Y 531.195,Z 1106.724,A -85,B 0,C 180,E1 4234.906,E2 4234.906} C_VEL
LIN {X 0,Y 531.384,Z 1096.648,A -85,B 0,C 180,E1 4238.604,E2 4238.604} C_VEL
LIN {X 0,Y 531.726,Z 1081.09,A -85,B 0,C 180,E1 4242.123,E2 4242.123} C_VEL
LIN {X 0,Y 532.561,Z 1059.671,A -85,B 0,C 180,E1 4245.459,E2 4245.459} C_VEL
LIN {X 0,Y 533.677,Z 1034.547,A -85,B 0,C 180,E1 4248.277,E2 4248.277} C_VEL
LIN {X 0,Y 535.026,Z 1005.075,A -85,B 0,C 180,E1 4250.647,E2 4250.647} C_VEL
LIN {X 0,Y 536.228,Z 972.398,A -85,B 0,C 180,E1 4252.462,E2 4252.462} C_VEL
LIN {X 0,Y 537.244,Z 937.831,A -85,B 0,C 180,E1 4253.645,E2 4253.645} C_VEL
LIN {X 0,Y 537.004,Z 876.314,A -85,B 0,C 180,E1 4254.649,E2 4254.649} C_VEL
LIN {X 0,Y 530.43,Z 857.28,A -85,B 0,C 180,E1 4255.352,E2 4255.352} C_VEL
LIN {X 0,Y 530.303,Z 857.28,A -85,B 0,C 180,E1 4261.071,E2 4261.071} C_VEL
LIN {X 0,Y 530.239,Z 857.28,A -85,B 0,C 180,E1 4266.913,E2 4266.913} C_VEL
LIN {X 0,Y 530.229,Z 857.28,A -85,B 0,C 180,E1 4273.262,E2 4273.262} C_VEL
LIN {X 0,Y 530.28,Z 857.28,A -85,B 0,C 180,E1 4278.945,E2 4278.945} C_VEL
LIN {X 0,Y 530.314,Z 857.28,A -85,B 0,C 180,E1 4285.171,E2 4285.171} C_VEL
LIN {X 0,Y 530.349,Z 857.28,A -85,B 0,C 180,E1 4290.956,E2 4290.956} C_VEL
LIN {X 0,Y 530.472,Z 857.28,A -85,B 0,C 180,E1 4296.436,E2 4296.436} C_VEL
LIN {X 0,Y 530.64,Z 857.28,A -85,B 0,C 180,E1 4301.694,E2 4301.694} C_VEL
LIN {X 0,Y 530.568,Z 857.28,A -85,B 0,C 180,E1 4308.461,E2 4308.461} C_VEL
LIN {X 0,Y 530.887,Z 857.28,A -85,B 0,C 180,E1 4313.431,E2 4313.431} C_VEL
LIN {X 0,Y 530.823,Z 857.28,A -85,B 0,C 180,E1 4319.979,E2 4319.979} C_VEL
LIN {X 0,Y 530.789,Z 857.28,A -85,B 0,C 180,E1 4324.886,E2 4324.886} C_VEL
LIN {X 0,Y 530.702,Z 857.28,A -85,B 0,C 180,E1 4329.831,E2 4329.831} C_VEL
LIN {X 0,Y 530.626,Z 857.28,A -85,B 0,C 180,E1 4334.852,E2 4334.852} C_VEL
LIN {X 0,Y 530.587,Z 857.28,A -85,B 0,C 180,E1 4339.994,E2 4339.994} C_VEL
LIN {X 0,Y 530.463,Z 857.28,A -85,B 0,C 180,E1 4345.315,E2 4345.315} C_VEL
LIN {X 0,Y 530.274,Z 857.28,A -85,B 0,C 180,E1 4351.064,E2 4351.064} C_VEL
LIN {X 0,Y 530.211,Z 857.28,A -85,B 0,C 180,E1 4356.91,E2 4356.91} C_VEL
LIN {X 0,Y 530.255,Z 857.28,A -85,B 0,C 180,E1 4363.206,E2 4363.206} C_VEL
LIN {X 0,Y 530.273,Z 857.28,A -85,B 0,C 180,E1 4368.949,E2 4368.949} C_VEL
LIN {X 0,Y 530.428,Z 857.28,A -85,B 0,C 180,E1 4375.187,E2 4375.187} C_VEL
LIN {X 0,Y 530.566,Z 858.071,A -85,B 0,C 180,E1 4376.657,E2 4376.657} C_VEL
LIN {X 0,Y 533.922,Z 876.205,A -85,B 0,C 180,E1 4377.653,E2 4377.653} C_VEL
LIN {X 0,Y 533.195,Z 901.352,A -85,B 0,C 180,E1 4379.381,E2 4379.381} C_VEL
LIN {X 0,Y 532.277,Z 923.321,A -85,B 0,C 180,E1 4381.635,E2 4381.635} C_VEL
